   1:  PR[91,1] = PR[90,1] + 6.641;
   1:  PR[91,2] = PR[90,2] + -29.893;
   1:  PR[91,3] = PR[90,3] + 98.074;
   1:L PR[91] R[100]mm/sec CNT100;
   1:  PR[91,1] = PR[90,1] + 10.896;
   1:  PR[91,2] = PR[90,2] + -30.120;
   1:  PR[91,3] = PR[90,3] + 98.081;
   1:L PR[91] R[100]mm/sec CNT100;
   1:  PR[91,1] = PR[90,1] + 16.041;
   1:  PR[91,2] = PR[90,2] + -30.372;
   1:  PR[91,3] = PR[90,3] + 98.101;
   1:L PR[91] R[100]mm/sec CNT100;
   1:  PR[91,1] = PR[90,1] + 18.590;
   1:  PR[91,2] = PR[90,2] + -30.271;
   1:  PR[91,3] = PR[90,3] + 98.125;
   1:L PR[91] R[100]mm/sec CNT100;
   1:  PR[91,1] = PR[90,1] + 25.648;
   1:  PR[91,2] = PR[90,2] + -29.896;
   1:  PR[91,3] = PR[90,3] + 98.137;
   1:L PR[91] R[100]mm/sec CNT100;
   1:  PR[91,1] = PR[90,1] + 25.448;
   1:  PR[91,2] = PR[90,2] + -30.607;
   1:  PR[91,3] = PR[90,3] + 98.169;
   1:L PR[91] R[100]mm/sec CNT100;
   1:  PR[91,1] = PR[90,1] + 28.784;
   1:  PR[91,2] = PR[90,2] + -31.148;
   1:  PR[91,3] = PR[90,3] + 98.173;
   1:L PR[91] R[100]mm/sec CNT100;
   1:  PR[91,1] = PR[90,1] + 29.348;
   1:  PR[91,2] = PR[90,2] + -31.179;
   1:  PR[91,3] = PR[90,3] + 98.188;
   1:L PR[91] R[100]mm/sec CNT100;
   1:  PR[91,1] = PR[90,1] + 34.258;
   1:  PR[91,2] = PR[90,2] + -31.084;
   1:  PR[91,3] = PR[90,3] + 98.191;
   1:L PR[91] R[100]mm/sec CNT100;
   1:  PR[91,1] = PR[90,1] + 35.080;
   1:  PR[91,2] = PR[90,2] + -30.981;
   1:  PR[91,3] = PR[90,3] + 98.214;
   1:L PR[91] R[100]mm/sec CNT100;
   1:  PR[91,1] = PR[90,1] + 39.542;
   1:  PR[91,2] = PR[90,2] + -30.057;
   1:  PR[91,3] = PR[90,3] + 98.217;
   1:L PR[91] R[100]mm/sec CNT100;
   1:  PR[91,1] = PR[90,1] + 40.641;
   1:  PR[91,2] = PR[90,2] + -29.713;
   1:  PR[91,3] = PR[90,3] + 98.239;
   1:L PR[91] R[100]mm/sec CNT100;
   1:  PR[91,1] = PR[90,1] + 44.461;
   1:  PR[91,2] = PR[90,2] + -28.152;
   1:  PR[91,3] = PR[90,3] + 98.244;
   1:L PR[91] R[100]mm/sec CNT100;
   1:  PR[91,1] = PR[90,1] + 45.821;
   1:  PR[91,2] = PR[90,2] + -27.441;
   1:  PR[91,3] = PR[90,3] + 98.263;
   1:L PR[91] R[100]mm/sec CNT100;
   1:  PR[91,1] = PR[90,1] + 48.863;
   1:  PR[91,2] = PR[90,2] + -25.483;
   1:  PR[91,3] = PR[90,3] + 98.270;
   1:L PR[91] R[100]mm/sec CNT100;
   1:  PR[91,1] = PR[90,1] + 50.435;
   1:  PR[91,2] = PR[90,2] + -24.267;
   1:  PR[91,3] = PR[90,3] + 98.287;
   1:L PR[91] R[100]mm/sec CNT100;
   1:  PR[91,1] = PR[90,1] + 52.635;
   1:  PR[91,2] = PR[90,2] + -22.198;
   1:  PR[91,3] = PR[90,3] + 98.296;
   1:L PR[91] R[100]mm/sec CNT100;
   1:  PR[91,1] = PR[90,1] + 54.323;
   1:  PR[91,2] = PR[90,2] + -20.343;
   1:  PR[91,3] = PR[90,3] + 98.310;
   1:L PR[91] R[100]mm/sec CNT100;
   1:  PR[91,1] = PR[90,1] + 55.712;
   1:  PR[91,2] = PR[90,2] + -18.450;
   1:  PR[91,3] = PR[90,3] + 98.321;
   1:L PR[91] R[100]mm/sec CNT100;
   1:  PR[91,1] = PR[90,1] + 57.371;
   1:  PR[91,2] = PR[90,2] + -15.845;
   1:  PR[91,3] = PR[90,3] + 98.332;
   1:L PR[91] R[100]mm/sec CNT100;
   1:  PR[91,1] = PR[90,1] + 58.087;
   1:  PR[91,2] = PR[90,2] + -14.370;
   1:  PR[91,3] = PR[90,3] + 98.347;
   1:L PR[91] R[100]mm/sec CNT100;
   1:  PR[91,1] = PR[90,1] + 59.526;
   1:  PR[91,2] = PR[90,2] + -10.971;
   1:  PR[91,3] = PR[90,3] + 98.354;
   1:L PR[91] R[100]mm/sec CNT100;
   1:  PR[91,1] = PR[90,1] + 59.787;
   1:  PR[91,2] = PR[90,2] + -10.029;
   1:  PR[91,3] = PR[90,3] + 98.371;
   1:L PR[91] R[100]mm/sec CNT100;
   1:  PR[91,1] = PR[90,1] + 60.788;
   1:  PR[91,2] = PR[90,2] + -5.902;
   1:  PR[91,3] = PR[90,3] + 98.376;
   1:L PR[91] R[100]mm/sec CNT100;
   1:  PR[91,1] = PR[90,1] + 61.174;
   1:  PR[91,2] = PR[90,2] + -1.109;
   1:  PR[91,3] = PR[90,3] + 98.395;
   1:L PR[91] R[100]mm/sec CNT100;
   1:  PR[91,1] = PR[90,1] + 61.192;
   1:  PR[91,2] = PR[90,2] + -0.755;
   1:  PR[91,3] = PR[90,3] + 98.418;
   1:L PR[91] R[100]mm/sec CNT100;
   1:  PR[91,1] = PR[90,1] + 60.788;
   1:  PR[91,2] = PR[90,2] + 4.445;
   1:  PR[91,3] = PR[90,3] + 98.419;
   1:L PR[91] R[100]mm/sec CNT100;
   1:  PR[91,1] = PR[90,1] + 59.787;
   1:  PR[91,2] = PR[90,2] + 8.570;
   1:  PR[91,3] = PR[90,3] + 98.443;
   1:L PR[91] R[100]mm/sec CNT100;
   1:  PR[91,1] = PR[90,1] + 59.526;
   1:  PR[91,2] = PR[90,2] + 9.512;
   1:  PR[91,3] = PR[90,3] + 98.463;
   1:L PR[91] R[100]mm/sec CNT100;
   1:  PR[91,1] = PR[90,1] + 58.087;
   1:  PR[91,2] = PR[90,2] + 12.910;
   1:  PR[91,3] = PR[90,3] + 98.467;
   1:L PR[91] R[100]mm/sec CNT100;
   1:  PR[91,1] = PR[90,1] + 57.372;
   1:  PR[91,2] = PR[90,2] + 14.385;
   1:  PR[91,3] = PR[90,3] + 98.484;
   1:L PR[91] R[100]mm/sec CNT100;
   1:  PR[91,1] = PR[90,1] + 55.713;
   1:  PR[91,2] = PR[90,2] + 16.990;
   1:  PR[91,3] = PR[90,3] + 98.492;
   1:L PR[91] R[100]mm/sec CNT100;
   1:  PR[91,1] = PR[90,1] + 54.325;
   1:  PR[91,2] = PR[90,2] + 18.882;
   1:  PR[91,3] = PR[90,3] + 98.506;
   1:L PR[91] R[100]mm/sec CNT100;
   1:  PR[91,1] = PR[90,1] + 52.637;
   1:  PR[91,2] = PR[90,2] + 20.737;
   1:  PR[91,3] = PR[90,3] + 98.517;
   1:L PR[91] R[100]mm/sec CNT100;
   1:  PR[91,1] = PR[90,1] + 50.438;
   1:  PR[91,2] = PR[90,2] + 22.806;
   1:  PR[91,3] = PR[90,3] + 98.529;
   1:L PR[91] R[100]mm/sec CNT100;
   1:  PR[91,1] = PR[90,1] + 48.866;
   1:  PR[91,2] = PR[90,2] + 24.022;
   1:  PR[91,3] = PR[90,3] + 98.543;
   1:L PR[91] R[100]mm/sec CNT100;
   1:  PR[91,1] = PR[90,1] + 45.826;
   1:  PR[91,2] = PR[90,2] + 25.979;
   1:  PR[91,3] = PR[90,3] + 98.552;
   1:L PR[91] R[100]mm/sec CNT100;
   1:  PR[91,1] = PR[90,1] + 44.466;
   1:  PR[91,2] = PR[90,2] + 26.691;
   1:  PR[91,3] = PR[90,3] + 98.569;
   1:L PR[91] R[100]mm/sec CNT100;
   1:  PR[91,1] = PR[90,1] + 40.648;
   1:  PR[91,2] = PR[90,2] + 28.252;
   1:  PR[91,3] = PR[90,3] + 98.576;
   1:L PR[91] R[100]mm/sec CNT100;
   1:  PR[91,1] = PR[90,1] + 39.550;
   1:  PR[91,2] = PR[90,2] + 28.596;
   1:  PR[91,3] = PR[90,3] + 98.595;
   1:L PR[91] R[100]mm/sec CNT100;
   1:  PR[91,1] = PR[90,1] + 35.089;
   1:  PR[91,2] = PR[90,2] + 29.521;
   1:  PR[91,3] = PR[90,3] + 98.600;
   1:L PR[91] R[100]mm/sec CNT100;
   1:  PR[91,1] = PR[90,1] + 34.267;
   1:  PR[91,2] = PR[90,2] + 29.624;
   1:  PR[91,3] = PR[90,3] + 98.621;
   1:L PR[91] R[100]mm/sec CNT100;
   1:  PR[91,1] = PR[90,1] + 29.359;
   1:  PR[91,2] = PR[90,2] + 29.721;
   1:  PR[91,3] = PR[90,3] + 98.625;
   1:L PR[91] R[100]mm/sec CNT100;
   1:  PR[91,1] = PR[90,1] + 28.796;
   1:  PR[91,2] = PR[90,2] + 29.690;
   1:  PR[91,3] = PR[90,3] + 98.648;
   1:L PR[91] R[100]mm/sec CNT100;
   1:  PR[91,1] = PR[90,1] + 23.729;
   1:  PR[91,2] = PR[90,2] + 28.869;
   1:  PR[91,3] = PR[90,3] + 98.650;
   1:L PR[91] R[100]mm/sec CNT100;
   1:  PR[91,1] = PR[90,1] + 23.140;
   1:  PR[91,2] = PR[90,2] + 28.730;
   1:  PR[91,3] = PR[90,3] + 98.674;
   1:L PR[91] R[100]mm/sec CNT100;
   1:  PR[91,1] = PR[90,1] + 18.623;
   1:  PR[91,2] = PR[90,2] + 28.811;
   1:  PR[91,3] = PR[90,3] + 98.677;
   1:L PR[91] R[100]mm/sec CNT100;
   1:  PR[91,1] = PR[90,1] + 16.042;
   1:  PR[91,2] = PR[90,2] + 28.913;
   1:  PR[91,3] = PR[90,3] + 98.698;
   1:L PR[91] R[100]mm/sec CNT100;
   1:  PR[91,1] = PR[90,1] + 10.897;
   1:  PR[91,2] = PR[90,2] + 28.661;
   1:  PR[91,3] = PR[90,3] + 98.710;
   1:L PR[91] R[100]mm/sec CNT100;
   1:  PR[91,1] = PR[90,1] + 6.641;
   1:  PR[91,2] = PR[90,2] + 28.434;
   1:  PR[91,3] = PR[90,3] + 98.733;
   1:L PR[91] R[100]mm/sec CNT100;
   1:  PR[91,1] = PR[90,1] + 5.106;
   1:  PR[91,2] = PR[90,2] + 28.225;
   1:  PR[91,3] = PR[90,3] + 98.753;
   1:L PR[91] R[100]mm/sec CNT100;
   1:  PR[91,1] = PR[90,1] + -3.145;
   1:  PR[91,2] = PR[90,2] + 27.325;
   1:  PR[91,3] = PR[90,3] + 98.760;
   1:L PR[91] R[100]mm/sec CNT100;
   1:  PR[91,1] = PR[90,1] + -5.199;
   1:  PR[91,2] = PR[90,2] + 26.959;
   1:  PR[91,3] = PR[90,3] + 98.799;
   1:L PR[91] R[100]mm/sec CNT100;
   1:  PR[91,1] = PR[90,1] + -12.780;
   1:  PR[91,2] = PR[90,2] + 25.572;
   1:  PR[91,3] = PR[90,3] + 98.808;
   1:L PR[91] R[100]mm/sec CNT100;
   1:  PR[91,1] = PR[90,1] + -16.949;
   1:  PR[91,2] = PR[90,2] + 24.489;
   1:  PR[91,3] = PR[90,3] + 98.844;
   1:L PR[91] R[100]mm/sec CNT100;
   1:  PR[91,1] = PR[90,1] + -21.539;
   1:  PR[91,2] = PR[90,2] + 23.273;
   1:  PR[91,3] = PR[90,3] + 98.864;
   1:L PR[91] R[100]mm/sec CNT100;
   1:  PR[91,1] = PR[90,1] + -29.296;
   1:  PR[91,2] = PR[90,2] + 20.506;
   1:  PR[91,3] = PR[90,3] + 98.886;
   1:L PR[91] R[100]mm/sec CNT100;
   1:  PR[91,1] = PR[90,1] + -35.940;
   1:  PR[91,2] = PR[90,2] + 17.361;
   1:  PR[91,3] = PR[90,3] + 98.924;
   1:L PR[91] R[100]mm/sec CNT100;
   1:  PR[91,1] = PR[90,1] + -38.987;
   1:  PR[91,2] = PR[90,2] + 15.439;
   1:  PR[91,3] = PR[90,3] + 98.958;
   1:L PR[91] R[100]mm/sec CNT100;
   1:  PR[91,1] = PR[90,1] + -41.065;
   1:  PR[91,2] = PR[90,2] + 14.002;
   1:  PR[91,3] = PR[90,3] + 98.974;
   1:L PR[91] R[100]mm/sec CNT100;
   1:  PR[91,1] = PR[90,1] + -42.431;
   1:  PR[91,2] = PR[90,2] + 12.638;
   1:  PR[91,3] = PR[90,3] + 98.986;
   1:L PR[91] R[100]mm/sec CNT100;
   1:  PR[91] = PR[90];
   1:  PR[91,1] = PR[90,1] + -44.925;
   1:  PR[91,2] = PR[90,2] + 7.871;
   1:  PR[91,3] = PR[90,3] + 100.295;
   1:L PR[91] R[100]mm/sec CNT100;
   1:  PR[91,1] = PR[90,1] + -46.371;
   1:  PR[91,2] = PR[90,2] + 5.287;
   1:  PR[91,3] = PR[90,3] + 99.008;
   1:L PR[91] R[100]mm/sec CNT100;
   1:  PR[91,1] = PR[90,1] + -46.992;
   1:  PR[91,2] = PR[90,2] + 3.826;
   1:  PR[91,3] = PR[90,3] + 99.021;
   1:L PR[91] R[100]mm/sec CNT100;
   1:  PR[91,1] = PR[90,1] + -47.631;
   1:  PR[91,2] = PR[90,2] + 0.359;
   1:  PR[91,3] = PR[90,3] + 99.029;
   1:L PR[91] R[100]mm/sec CNT100;
   1:  PR[91,1] = PR[90,1] + -47.771;
   1:  PR[91,2] = PR[90,2] + -0.655;
   1:  PR[91,3] = PR[90,3] + 99.045;
   1:L PR[91] R[100]mm/sec CNT100;
   1:  PR[91,1] = PR[90,1] + -47.136;
   1:  PR[91,2] = PR[90,2] + -3.623;
   1:  PR[91,3] = PR[90,3] + 99.050;
   1:L PR[91] R[100]mm/sec CNT100;
   1:  PR[91,1] = PR[90,1] + -46.916;
   1:  PR[91,2] = PR[90,2] + -5.255;
   1:  PR[91,3] = PR[90,3] + 99.064;
   1:L PR[91] R[100]mm/sec CNT100;
   1:  PR[91,1] = PR[90,1] + -46.201;
   1:  PR[91,2] = PR[90,2] + -6.956;
   1:  PR[91,3] = PR[90,3] + 99.072;
   1:L PR[91] R[100]mm/sec CNT100;
   1:  PR[91,1] = PR[90,1] + -44.928;
   1:  PR[91,2] = PR[90,2] + -9.234;
   1:  PR[91,3] = PR[90,3] + 99.081;
   1:L PR[91] R[100]mm/sec CNT100;
   1:  PR[91,1] = PR[90,1] + -43.216;
   1:  PR[91,2] = PR[90,2] + -11.609;
   1:  PR[91,3] = PR[90,3] + 99.093;
   1:L PR[91] R[100]mm/sec CNT100;
   1:  PR[91,1] = PR[90,1] + -42.222;
   1:  PR[91,2] = PR[90,2] + -12.617;
   1:  PR[91,3] = PR[90,3] + 99.106;
   1:L PR[91] R[100]mm/sec CNT100;
   1:  PR[91,1] = PR[90,1] + -39.392;
   1:  PR[91,2] = PR[90,2] + -15.330;
   1:  PR[91,3] = PR[90,3] + 99.113;
   1:L PR[91] R[100]mm/sec CNT100;
   1:  PR[91,1] = PR[90,1] + -39.188;
   1:  PR[91,2] = PR[90,2] + -15.505;
   1:  PR[91,3] = PR[90,3] + 99.131;
   1:L PR[91] R[100]mm/sec CNT100;
   1:  PR[91,1] = PR[90,1] + -33.702;
   1:  PR[91,2] = PR[90,2] + -18.967;
   1:  PR[91,3] = PR[90,3] + 99.133;
   1:L PR[91] R[100]mm/sec CNT100;
   1:  PR[91,1] = PR[90,1] + -27.011;
   1:  PR[91,2] = PR[90,2] + -22.137;
   1:  PR[91,3] = PR[90,3] + 99.163;
   1:L PR[91] R[100]mm/sec CNT100;
   1:  PR[91,1] = PR[90,1] + -19.200;
   1:  PR[91,2] = PR[90,2] + -24.928;
   1:  PR[91,3] = PR[90,3] + 99.197;
   1:L PR[91] R[100]mm/sec CNT100;
   1:  PR[91,1] = PR[90,1] + -13.832;
   1:  PR[91,2] = PR[90,2] + -26.349;
   1:  PR[91,3] = PR[90,3] + 99.236;
   1:L PR[91] R[100]mm/sec CNT100;
   1:  PR[91,1] = PR[90,1] + -10.380;
   1:  PR[91,2] = PR[90,2] + -27.246;
   1:  PR[91,3] = PR[90,3] + 99.262;
   1:L PR[91] R[100]mm/sec CNT100;
   1:  PR[91,1] = PR[90,1] + -0.670;
   1:  PR[91,2] = PR[90,2] + -29.016;
   1:  PR[91,3] = PR[90,3] + 99.279;
   1:L PR[91] R[100]mm/sec CNT100;
   1:  PR[91,1] = PR[90,1] + 4.458;
   1:  PR[91,2] = PR[90,2] + -29.576;
   1:  PR[91,3] = PR[90,3] + 99.325;
   1:L PR[91] R[100]mm/sec CNT100;
   1:  PR[91,1] = PR[90,1] + 8.317;
   1:  PR[91,2] = PR[90,2] + -30.101;
   1:  PR[91,3] = PR[90,3] + 99.349;
   1:L PR[91] R[100]mm/sec CNT100;
   1:  PR[91,1] = PR[90,1] + 18.123;
   1:  PR[91,2] = PR[90,2] + -30.626;
   1:  PR[91,3] = PR[90,3] + 99.367;
   1:L PR[91] R[100]mm/sec CNT100;
   1:  PR[91,1] = PR[90,1] + 26.250;
   1:  PR[91,2] = PR[90,2] + -30.195;
   1:  PR[91,3] = PR[90,3] + 99.413;
   1:L PR[91] R[100]mm/sec CNT100;
   1:  PR[91,1] = PR[90,1] + 26.060;
   1:  PR[91,2] = PR[90,2] + -30.872;
   1:  PR[91,3] = PR[90,3] + 99.451;
   1:L PR[91] R[100]mm/sec CNT100;
   1:  PR[91,1] = PR[90,1] + 28.993;
   1:  PR[91,2] = PR[90,2] + -31.346;
   1:  PR[91,3] = PR[90,3] + 99.454;
   1:L PR[91] R[100]mm/sec CNT100;
   1:  PR[91,1] = PR[90,1] + 34.620;
   1:  PR[91,2] = PR[90,2] + -31.231;
   1:  PR[91,3] = PR[90,3] + 99.468;
   1:L PR[91] R[100]mm/sec CNT100;
   1:  PR[91,1] = PR[90,1] + 40.124;
   1:  PR[91,2] = PR[90,2] + -30.092;
   1:  PR[91,3] = PR[90,3] + 99.494;
   1:L PR[91] R[100]mm/sec CNT100;
   1:  PR[91,1] = PR[90,1] + 40.146;
   1:  PR[91,2] = PR[90,2] + -30.085;
   1:  PR[91,3] = PR[90,3] + 99.521;
   1:L PR[91] R[100]mm/sec CNT100;
   1:  PR[91,1] = PR[90,1] + 45.193;
   1:  PR[91,2] = PR[90,2] + -28.023;
   1:L PR[91] R[100]mm/sec CNT100;
   1:  PR[91,1] = PR[90,1] + 45.424;
   1:  PR[91,2] = PR[90,2] + -27.902;
   1:  PR[91,3] = PR[90,3] + 99.546;
   1:L PR[91] R[100]mm/sec CNT100;
   1:  PR[91,1] = PR[90,1] + 49.743;
   1:  PR[91,2] = PR[90,2] + -25.122;
   1:  PR[91,3] = PR[90,3] + 99.547;
   1:L PR[91] R[100]mm/sec CNT100;
   1:  PR[91,1] = PR[90,1] + 50.169;
   1:  PR[91,2] = PR[90,2] + -24.793;
   1:  PR[91,3] = PR[90,3] + 99.571;
   1:L PR[91] R[100]mm/sec CNT100;
   1:  PR[91,1] = PR[90,1] + 53.644;
   1:  PR[91,2] = PR[90,2] + -21.525;
   1:  PR[91,3] = PR[90,3] + 99.574;
   1:L PR[91] R[100]mm/sec CNT100;
   1:  PR[91,1] = PR[90,1] + 54.218;
   1:  PR[91,2] = PR[90,2] + -20.895;
   1:  PR[91,3] = PR[90,3] + 99.596;
   1:L PR[91] R[100]mm/sec CNT100;
   1:  PR[91,1] = PR[90,1] + 56.802;
   1:  PR[91,2] = PR[90,2] + -17.374;
   1:  PR[91,3] = PR[90,3] + 99.600;
   1:L PR[91] R[100]mm/sec CNT100;
   1:  PR[91,1] = PR[90,1] + 57.445;
   1:  PR[91,2] = PR[90,2] + -16.364;
   1:  PR[91,3] = PR[90,3] + 99.620;
   1:L PR[91] R[100]mm/sec CNT100;
   1:  PR[91,1] = PR[90,1] + 59.170;
   1:  PR[91,2] = PR[90,2] + -12.806;
   1:  PR[91,3] = PR[90,3] + 99.626;
   1:L PR[91] R[100]mm/sec CNT100;
   1:  PR[91,1] = PR[90,1] + 59.773;
   1:  PR[91,2] = PR[90,2] + -11.383;
   1:  PR[91,3] = PR[90,3] + 99.645;
   1:L PR[91] R[100]mm/sec CNT100;
   1:  PR[91,1] = PR[90,1] + 60.727;
   1:  PR[91,2] = PR[90,2] + -7.931;
   1:  PR[91,3] = PR[90,3] + 99.652;
   1:L PR[91] R[100]mm/sec CNT100;
   1:  PR[91,1] = PR[90,1] + 61.163;
   1:  PR[91,2] = PR[90,2] + -6.135;
   1:  PR[91,3] = PR[90,3] + 99.668;
   1:L PR[91] R[100]mm/sec CNT100;
   1:  PR[91,1] = PR[90,1] + 61.350;
   1:  PR[91,2] = PR[90,2] + -3.722;
   1:  PR[91,3] = PR[90,3] + 99.677;
   1:L PR[91] R[100]mm/sec CNT100;
   1:  PR[91,1] = PR[90,1] + 61.612;
   1:  PR[91,2] = PR[90,2] + -0.718;
   1:  PR[91,3] = PR[90,3] + 99.688;
   1:L PR[91] R[100]mm/sec CNT100;
   1:  PR[91,1] = PR[90,1] + 61.475;
   1:  PR[91,2] = PR[90,2] + 1.093;
   1:  PR[91,3] = PR[90,3] + 99.702;
   1:L PR[91] R[100]mm/sec CNT100;
   1:  PR[91,1] = PR[90,1] + 61.166;
   1:  PR[91,2] = PR[90,2] + 4.666;
   1:  PR[91,3] = PR[90,3] + 99.711;
   1:L PR[91] R[100]mm/sec CNT100;
   1:  PR[91,1] = PR[90,1] + 60.727;
   1:  PR[91,2] = PR[90,2] + 6.472;
   1:  PR[91,3] = PR[90,3] + 99.728;
   1:L PR[91] R[100]mm/sec CNT100;
   1:  PR[91,1] = PR[90,1] + 59.774;
   1:  PR[91,2] = PR[90,2] + 9.922;
   1:  PR[91,3] = PR[90,3] + 99.736;
   1:L PR[91] R[100]mm/sec CNT100;
   1:  PR[91,1] = PR[90,1] + 59.171;
   1:  PR[91,2] = PR[90,2] + 11.346;
   1:  PR[91,3] = PR[90,3] + 99.753;
   1:L PR[91] R[100]mm/sec CNT100;
   1:  PR[91,1] = PR[90,1] + 57.446;
   1:  PR[91,2] = PR[90,2] + 14.902;
   1:  PR[91,3] = PR[90,3] + 99.760;
   1:L PR[91] R[100]mm/sec CNT100;
   1:  PR[91,1] = PR[90,1] + 56.803;
   1:  PR[91,2] = PR[90,2] + 15.912;
   1:  PR[91,3] = PR[90,3] + 99.779;
   1:L PR[91] R[100]mm/sec CNT100;
   1:  PR[91,1] = PR[90,1] + 54.221;
   1:  PR[91,2] = PR[90,2] + 19.433;
   1:  PR[91,3] = PR[90,3] + 99.784;
   1:L PR[91] R[100]mm/sec CNT100;
   1:  PR[91,1] = PR[90,1] + 53.647;
   1:  PR[91,2] = PR[90,2] + 20.063;
   1:  PR[91,3] = PR[90,3] + 99.805;
   1:L PR[91] R[100]mm/sec CNT100;
   1:  PR[91,1] = PR[90,1] + 50.174;
   1:  PR[91,2] = PR[90,2] + 23.330;
   1:  PR[91,3] = PR[90,3] + 99.809;
   1:L PR[91] R[100]mm/sec CNT100;
   1:  PR[91,1] = PR[90,1] + 49.748;
   1:  PR[91,2] = PR[90,2] + 23.660;
   1:  PR[91,3] = PR[90,3] + 99.831;
   1:L PR[91] R[100]mm/sec CNT100;
   1:  PR[91,1] = PR[90,1] + 45.431;
   1:  PR[91,2] = PR[90,2] + 26.439;
   1:  PR[91,3] = PR[90,3] + 99.833;
   1:L PR[91] R[100]mm/sec CNT100;
   1:  PR[91,1] = PR[90,1] + 45.200;
   1:  PR[91,2] = PR[90,2] + 26.560;
   1:  PR[91,3] = PR[90,3] + 99.857;
   1:L PR[91] R[100]mm/sec CNT100;
   1:  PR[91,1] = PR[90,1] + 40.155;
   1:  PR[91,2] = PR[90,2] + 28.623;
   1:  PR[91,3] = PR[90,3] + 99.859;
   1:L PR[91] R[100]mm/sec CNT100;
   1:  PR[91,1] = PR[90,1] + 40.133;
   1:  PR[91,2] = PR[90,2] + 28.630;
   1:  PR[91,3] = PR[90,3] + 99.884;
   1:L PR[91] R[100]mm/sec CNT100;
   1:  PR[91,1] = PR[90,1] + 34.626;
   1:  PR[91,2] = PR[90,2] + 29.771;
   1:L PR[91] R[100]mm/sec CNT100;
   1:  PR[91,1] = PR[90,1] + 29.012;
   1:  PR[91,2] = PR[90,2] + 29.888;
   1:  PR[91,3] = PR[90,3] + 99.910;
   1:L PR[91] R[100]mm/sec CNT100;
   1:  PR[91,1] = PR[90,1] + 28.964;
   1:  PR[91,2] = PR[90,2] + 29.884;
   1:  PR[91,3] = PR[90,3] + 99.937;
   1:L PR[91] R[100]mm/sec CNT100;
   1:  PR[91,1] = PR[90,1] + 23.663;
   1:  PR[91,2] = PR[90,2] + 29.025;
   1:L PR[91] R[100]mm/sec CNT100;
   1:  PR[91,1] = PR[90,1] + 18.121;
   1:  PR[91,2] = PR[90,2] + 29.168;
   1:  PR[91,3] = PR[90,3] + 99.962;
   1:L PR[91] R[100]mm/sec CNT100;
   1:  PR[91,1] = PR[90,1] + 8.318;
   1:  PR[91,2] = PR[90,2] + 28.642;
   1:  PR[91,3] = PR[90,3] + 99.988;
   1:L PR[91] R[100]mm/sec CNT100;
   1:  PR[91,1] = PR[90,1] + 4.458;
   1:  PR[91,2] = PR[90,2] + 28.117;
   1:  PR[91,3] = PR[90,3] + 100.034;
   1:L PR[91] R[100]mm/sec CNT100;
   1:  PR[91,1] = PR[90,1] + -0.670;
   1:  PR[91,2] = PR[90,2] + 27.557;
   1:  PR[91,3] = PR[90,3] + 100.052;
   1:L PR[91] R[100]mm/sec CNT100;
   1:  PR[91,1] = PR[90,1] + -10.380;
   1:  PR[91,2] = PR[90,2] + 25.788;
   1:  PR[91,3] = PR[90,3] + 100.076;
   1:L PR[91] R[100]mm/sec CNT100;
   1:  PR[91,1] = PR[90,1] + -13.831;
   1:  PR[91,2] = PR[90,2] + 24.891;
   1:  PR[91,3] = PR[90,3] + 100.122;
   1:L PR[91] R[100]mm/sec CNT100;
   1:  PR[91,1] = PR[90,1] + -19.200;
   1:  PR[91,2] = PR[90,2] + 23.469;
   1:  PR[91,3] = PR[90,3] + 100.139;
   1:L PR[91] R[100]mm/sec CNT100;
   1:  PR[91,1] = PR[90,1] + -27.011;
   1:  PR[91,2] = PR[90,2] + 20.679;
   1:  PR[91,3] = PR[90,3] + 100.165;
   1:L PR[91] R[100]mm/sec CNT100;
   1:  PR[91,1] = PR[90,1] + -33.702;
   1:  PR[91,2] = PR[90,2] + 17.508;
   1:  PR[91,3] = PR[90,3] + 100.203;
   1:L PR[91] R[100]mm/sec CNT100;
   1:  PR[91,1] = PR[90,1] + -39.188;
   1:  PR[91,2] = PR[90,2] + 14.047;
   1:  PR[91,3] = PR[90,3] + 100.238;
   1:L PR[91] R[100]mm/sec CNT100;
   1:  PR[91,1] = PR[90,1] + -39.388;
   1:  PR[91,2] = PR[90,2] + 13.874;
   1:  PR[91,3] = PR[90,3] + 100.268;
   1:L PR[91] R[100]mm/sec CNT100;
   1:  PR[91,1] = PR[90,1] + -43.328;
   1:  PR[91,2] = PR[90,2] + 10.061;
   1:  PR[91,3] = PR[90,3] + 100.269;
   1:L PR[91] R[100]mm/sec CNT100;
   1:  PR[91] = PR[90];
   1:  PR[91,1] = PR[90,1] + -43.344;
   1:  PR[91,2] = PR[90,2] + 7.465;
   1:  PR[91,3] = PR[90,3] + 101.595;
   1:L PR[91] R[100]mm/sec CNT100;
   1:  PR[91,1] = PR[90,1] + -44.199;
   1:  PR[91,2] = PR[90,2] + 5.937;
   1:  PR[91,3] = PR[90,3] + 100.312;
   1:L PR[91] R[100]mm/sec CNT100;
   1:  PR[91,1] = PR[90,1] + -45.194;
   1:  PR[91,2] = PR[90,2] + 3.593;
   1:  PR[91,3] = PR[90,3] + 100.321;
   1:L PR[91] R[100]mm/sec CNT100;
   1:  PR[91,1] = PR[90,1] + -45.628;
   1:  PR[91,2] = PR[90,2] + 1.240;
   1:  PR[91,3] = PR[90,3] + 100.333;
   1:L PR[91] R[100]mm/sec CNT100;
   1:  PR[91,1] = PR[90,1] + -45.891;
   1:  PR[91,2] = PR[90,2] + -0.655;
   1:  PR[91,3] = PR[90,3] + 100.344;
   1:L PR[91] R[100]mm/sec CNT100;
   1:  PR[91,1] = PR[90,1] + -45.449;
   1:  PR[91,2] = PR[90,2] + -2.720;
   1:  PR[91,3] = PR[90,3] + 100.353;
   1:L PR[91] R[100]mm/sec CNT100;
   1:  PR[91,1] = PR[90,1] + -45.135;
   1:  PR[91,2] = PR[90,2] + -5.045;
   1:  PR[91,3] = PR[90,3] + 100.363;
   1:L PR[91] R[100]mm/sec CNT100;
   1:  PR[91,1] = PR[90,1] + -44.092;
   1:  PR[91,2] = PR[90,2] + -7.528;
   1:  PR[91,3] = PR[90,3] + 100.374;
   1:L PR[91] R[100]mm/sec CNT100;
   1:  PR[91,1] = PR[90,1] + -43.344;
   1:  PR[91,2] = PR[90,2] + -8.866;
   1:  PR[91,3] = PR[90,3] + 100.387;
   1:L PR[91] R[100]mm/sec CNT100;
   1:  PR[91,1] = PR[90,1] + -41.134;
   1:  PR[91,2] = PR[90,2] + -11.932;
   1:  PR[91,3] = PR[90,3] + 100.394;
   1:L PR[91] R[100]mm/sec CNT100;
   1:  PR[91,1] = PR[90,1] + -40.904;
   1:  PR[91,2] = PR[90,2] + -12.166;
   1:  PR[91,3] = PR[90,3] + 100.412;
   1:L PR[91] R[100]mm/sec CNT100;
   1:  PR[91,1] = PR[90,1] + -40.040;
   1:  PR[91,2] = PR[90,2] + -12.993;
   1:  PR[91,3] = PR[90,3] + 100.413;
   1:L PR[91] R[100]mm/sec CNT100;
   1:  PR[91,1] = PR[90,1] + -36.989;
   1:  PR[91,2] = PR[90,2] + -15.626;
   1:  PR[91,3] = PR[90,3] + 100.419;
   1:L PR[91] R[100]mm/sec CNT100;
   1:  PR[91,1] = PR[90,1] + -31.464;
   1:  PR[91,2] = PR[90,2] + -19.115;
   1:  PR[91,3] = PR[90,3] + 100.438;
   1:L PR[91] R[100]mm/sec CNT100;
   1:  PR[91,1] = PR[90,1] + -24.726;
   1:  PR[91,2] = PR[90,2] + -22.310;
   1:  PR[91,3] = PR[90,3] + 100.469;
   1:L PR[91] R[100]mm/sec CNT100;
   1:  PR[91,1] = PR[90,1] + -16.862;
   1:  PR[91,2] = PR[90,2] + -25.123;
   1:  PR[91,3] = PR[90,3] + 100.504;
   1:L PR[91] R[100]mm/sec CNT100;
   1:  PR[91,1] = PR[90,1] + -7.975;
   1:  PR[91,2] = PR[90,2] + -27.463;
   1:  PR[91,3] = PR[90,3] + 100.543;
   1:L PR[91] R[100]mm/sec CNT100;
   1:  PR[91,1] = PR[90,1] + 1.801;
   1:  PR[91,2] = PR[90,2] + -29.248;
   1:  PR[91,3] = PR[90,3] + 100.586;
   1:L PR[91] R[100]mm/sec CNT100;
   1:  PR[91,1] = PR[90,1] + 3.810;
   1:  PR[91,2] = PR[90,2] + -29.467;
   1:  PR[91,3] = PR[90,3] + 100.633;
   1:L PR[91] R[100]mm/sec CNT100;
   1:  PR[91,1] = PR[90,1] + 9.993;
   1:  PR[91,2] = PR[90,2] + -30.309;
   1:  PR[91,3] = PR[90,3] + 100.643;
   1:L PR[91] R[100]mm/sec CNT100;
   1:  PR[91,1] = PR[90,1] + 17.071;
   1:  PR[91,2] = PR[90,2] + -30.686;
   1:  PR[91,3] = PR[90,3] + 100.672;
   1:L PR[91] R[100]mm/sec CNT100;
   1:  PR[91,1] = PR[90,1] + 19.711;
   1:  PR[91,2] = PR[90,2] + -30.859;
   1:  PR[91,3] = PR[90,3] + 100.706;
   1:L PR[91] R[100]mm/sec CNT100;
   1:  PR[91,1] = PR[90,1] + 19.899;
   1:  PR[91,2] = PR[90,2] + -30.862;
   1:  PR[91,3] = PR[90,3] + 100.718;
   1:L PR[91] R[100]mm/sec CNT100;
   1:  PR[91,1] = PR[90,1] + 26.852;
   1:  PR[91,2] = PR[90,2] + -30.493;
   1:  PR[91,3] = PR[90,3] + 100.719;
   1:L PR[91] R[100]mm/sec CNT100;
   1:  PR[91,1] = PR[90,1] + 26.671;
   1:  PR[91,2] = PR[90,2] + -31.138;
   1:  PR[91,3] = PR[90,3] + 100.752;
   1:L PR[91] R[100]mm/sec CNT100;
   1:  PR[91,1] = PR[90,1] + 28.452;
   1:  PR[91,2] = PR[90,2] + -31.427;
   1:  PR[91,3] = PR[90,3] + 100.755;
   1:L PR[91] R[100]mm/sec CNT100;
   1:  PR[91,1] = PR[90,1] + 28.695;
   1:  PR[91,2] = PR[90,2] + -31.455;
   1:  PR[91,3] = PR[90,3] + 100.764;
   1:L PR[91] R[100]mm/sec CNT100;
   1:  PR[91,1] = PR[90,1] + 29.671;
   1:  PR[91,2] = PR[90,2] + -31.519;
   1:  PR[91,3] = PR[90,3] + 100.765;
   1:L PR[91] R[100]mm/sec CNT100;
   1:  PR[91,1] = PR[90,1] + 34.356;
   1:  PR[91,2] = PR[90,2] + -31.423;
   1:  PR[91,3] = PR[90,3] + 100.769;
   1:L PR[91] R[100]mm/sec CNT100;
   1:  PR[91,1] = PR[90,1] + 35.246;
   1:  PR[91,2] = PR[90,2] + -31.332;
   1:  PR[91,3] = PR[90,3] + 100.791;
   1:L PR[91] R[100]mm/sec CNT100;
   1:  PR[91,1] = PR[90,1] + 39.887;
   1:  PR[91,2] = PR[90,2] + -30.361;
   1:  PR[91,3] = PR[90,3] + 100.796;
   1:L PR[91] R[100]mm/sec CNT100;
   1:  PR[91,1] = PR[90,1] + 40.682;
   1:  PR[91,2] = PR[90,2] + -30.139;
   1:  PR[91,3] = PR[90,3] + 100.818;
   1:L PR[91] R[100]mm/sec CNT100;
   1:  PR[91,1] = PR[90,1] + 45.128;
   1:  PR[91,2] = PR[90,2] + -28.305;
   1:  PR[91,3] = PR[90,3] + 100.822;
   1:L PR[91] R[100]mm/sec CNT100;
   1:  PR[91,1] = PR[90,1] + 45.801;
   1:  PR[91,2] = PR[90,2] + -27.987;
   1:  PR[91,3] = PR[90,3] + 100.845;
   1:L PR[91] R[100]mm/sec CNT100;
   1:  PR[91,1] = PR[90,1] + 49.908;
   1:  PR[91,2] = PR[90,2] + -25.320;
   1:  PR[91,3] = PR[90,3] + 100.848;
   1:L PR[91] R[100]mm/sec CNT100;
   1:  PR[91,1] = PR[90,1] + 50.441;
   1:  PR[91,2] = PR[90,2] + -24.946;
   1:  PR[91,3] = PR[90,3] + 100.871;
   1:L PR[91] R[100]mm/sec CNT100;
   1:  PR[91,1] = PR[90,1] + 54.067;
   1:  PR[91,2] = PR[90,2] + -21.507;
   1:  PR[91,3] = PR[90,3] + 100.874;
   1:L PR[91] R[100]mm/sec CNT100;
   1:  PR[91,1] = PR[90,1] + 54.453;
   1:  PR[91,2] = PR[90,2] + -21.125;
   1:  PR[91,3] = PR[90,3] + 100.898;
   1:L PR[91] R[100]mm/sec CNT100;
   1:  PR[91,1] = PR[90,1] + 57.716;
   1:  PR[91,2] = PR[90,2] + -16.629;
   1:  PR[91,3] = PR[90,3] + 100.900;
   1:L PR[91] R[100]mm/sec CNT100;
   1:  PR[91,1] = PR[90,1] + 60.117;
   1:  PR[91,2] = PR[90,2] + -11.632;
   1:  PR[91,3] = PR[90,3] + 100.927;
   1:L PR[91] R[100]mm/sec CNT100;
   1:  PR[91,1] = PR[90,1] + 61.589;
   1:  PR[91,2] = PR[90,2] + -6.270;
   1:  PR[91,3] = PR[90,3] + 100.953;
   1:L PR[91] R[100]mm/sec CNT100;
   1:  PR[91,1] = PR[90,1] + 62.101;
   1:  PR[91,2] = PR[90,2] + -0.729;
   1:  PR[91,3] = PR[90,3] + 100.979;
   1:L PR[91] R[100]mm/sec CNT100;
   1:  PR[91,1] = PR[90,1] + 61.589;
   1:  PR[91,2] = PR[90,2] + 4.810;
   1:  PR[91,3] = PR[90,3] + 101.005;
   1:L PR[91] R[100]mm/sec CNT100;
   1:  PR[91,1] = PR[90,1] + 60.117;
   1:  PR[91,2] = PR[90,2] + 10.174;
   1:  PR[91,3] = PR[90,3] + 101.031;
   1:L PR[91] R[100]mm/sec CNT100;
   1:  PR[91,1] = PR[90,1] + 59.976;
   1:  PR[91,2] = PR[90,2] + 10.471;
   1:  PR[91,3] = PR[90,3] + 101.058;
   1:L PR[91] R[100]mm/sec CNT100;
   1:  PR[91,1] = PR[90,1] + 57.718;
   1:  PR[91,2] = PR[90,2] + 15.167;
   1:  PR[91,3] = PR[90,3] + 101.059;
   1:L PR[91] R[100]mm/sec CNT100;
   1:  PR[91,1] = PR[90,1] + 54.455;
   1:  PR[91,2] = PR[90,2] + 19.663;
   1:  PR[91,3] = PR[90,3] + 101.084;
   1:L PR[91] R[100]mm/sec CNT100;
   1:  PR[91,1] = PR[90,1] + 54.070;
   1:  PR[91,2] = PR[90,2] + 20.045;
   1:  PR[91,3] = PR[90,3] + 101.110;
   1:L PR[91] R[100]mm/sec CNT100;
   1:  PR[91,1] = PR[90,1] + 50.445;
   1:  PR[91,2] = PR[90,2] + 23.485;
   1:  PR[91,3] = PR[90,3] + 101.112;
   1:L PR[91] R[100]mm/sec CNT100;
   1:  PR[91,1] = PR[90,1] + 49.912;
   1:  PR[91,2] = PR[90,2] + 23.858;
   1:  PR[91,3] = PR[90,3] + 101.136;
   1:L PR[91] R[100]mm/sec CNT100;
   1:  PR[91,1] = PR[90,1] + 45.805;
   1:  PR[91,2] = PR[90,2] + 26.526;
   1:  PR[91,3] = PR[90,3] + 101.139;
   1:L PR[91] R[100]mm/sec CNT100;
   1:  PR[91,1] = PR[90,1] + 45.133;
   1:  PR[91,2] = PR[90,2] + 26.844;
   1:  PR[91,3] = PR[90,3] + 101.162;
   1:L PR[91] R[100]mm/sec CNT100;
   1:  PR[91,1] = PR[90,1] + 40.687;
   1:  PR[91,2] = PR[90,2] + 28.679;
   1:  PR[91,3] = PR[90,3] + 101.166;
   1:L PR[91] R[100]mm/sec CNT100;
   1:  PR[91,1] = PR[90,1] + 39.892;
   1:  PR[91,2] = PR[90,2] + 28.900;
   1:  PR[91,3] = PR[90,3] + 101.188;
   1:L PR[91] R[100]mm/sec CNT100;
   1:  PR[91,1] = PR[90,1] + 35.251;
   1:  PR[91,2] = PR[90,2] + 29.873;
   1:  PR[91,3] = PR[90,3] + 101.192;
   1:L PR[91] R[100]mm/sec CNT100;
   1:  PR[91,1] = PR[90,1] + 34.362;
   1:  PR[91,2] = PR[90,2] + 29.964;
   1:  PR[91,3] = PR[90,3] + 101.215;
   1:L PR[91] R[100]mm/sec CNT100;
   1:  PR[91,1] = PR[90,1] + 29.677;
   1:  PR[91,2] = PR[90,2] + 30.061;
   1:  PR[91,3] = PR[90,3] + 101.219;
   1:L PR[91] R[100]mm/sec CNT100;
   1:  PR[91,1] = PR[90,1] + 28.703;
   1:  PR[91,2] = PR[90,2] + 29.996;
   1:  PR[91,3] = PR[90,3] + 101.241;
   1:L PR[91] R[100]mm/sec CNT100;
   1:  PR[91,1] = PR[90,1] + 28.411;
   1:  PR[91,2] = PR[90,2] + 29.962;
   1:  PR[91,3] = PR[90,3] + 101.245;
   1:L PR[91] R[100]mm/sec CNT100;
   1:  PR[91,1] = PR[90,1] + 24.273;
   1:  PR[91,2] = PR[90,2] + 29.292;
   1:  PR[91,3] = PR[90,3] + 101.247;
   1:L PR[91] R[100]mm/sec CNT100;
   1:  PR[91,1] = PR[90,1] + 19.975;
   1:  PR[91,2] = PR[90,2] + 29.404;
   1:  PR[91,3] = PR[90,3] + 101.267;
   1:L PR[91] R[100]mm/sec CNT100;
   1:  PR[91,1] = PR[90,1] + 19.713;
   1:  PR[91,2] = PR[90,2] + 29.400;
   1:  PR[91,3] = PR[90,3] + 101.287;
   1:L PR[91] R[100]mm/sec CNT100;
   1:  PR[91,1] = PR[90,1] + 17.071;
   1:  PR[91,2] = PR[90,2] + 29.227;
   1:  PR[91,3] = PR[90,3] + 101.288;
   1:L PR[91] R[100]mm/sec CNT100;
   1:  PR[91,1] = PR[90,1] + 9.994;
   1:  PR[91,2] = PR[90,2] + 28.850;
   1:  PR[91,3] = PR[90,3] + 101.301;
   1:L PR[91] R[100]mm/sec CNT100;
   1:  PR[91,1] = PR[90,1] + 3.810;
   1:  PR[91,2] = PR[90,2] + 28.009;
   1:  PR[91,3] = PR[90,3] + 101.334;
   1:L PR[91] R[100]mm/sec CNT100;
   1:  PR[91,1] = PR[90,1] + 1.801;
   1:  PR[91,2] = PR[90,2] + 27.789;
   1:  PR[91,3] = PR[90,3] + 101.363;
   1:L PR[91] R[100]mm/sec CNT100;
   1:  PR[91,1] = PR[90,1] + -7.978;
   1:  PR[91,2] = PR[90,2] + 26.003;
   1:  PR[91,3] = PR[90,3] + 101.373;
   1:L PR[91] R[100]mm/sec CNT100;
   1:  PR[91,1] = PR[90,1] + -10.714;
   1:  PR[91,2] = PR[90,2] + 25.292;
   1:  PR[91,3] = PR[90,3] + 101.420;
   1:L PR[91] R[100]mm/sec CNT100;
   1:  PR[91,1] = PR[90,1] + -16.860;
   1:  PR[91,2] = PR[90,2] + 23.665;
   1:  PR[91,3] = PR[90,3] + 101.433;
   1:L PR[91] R[100]mm/sec CNT100;
   1:  PR[91,1] = PR[90,1] + -24.726;
   1:  PR[91,2] = PR[90,2] + 20.852;
   1:  PR[91,3] = PR[90,3] + 101.463;
   1:L PR[91] R[100]mm/sec CNT100;
   1:  PR[91,1] = PR[90,1] + -31.465;
   1:  PR[91,2] = PR[90,2] + 17.656;
   1:  PR[91,3] = PR[90,3] + 101.503;
   1:L PR[91] R[100]mm/sec CNT100;
   1:  PR[91,1] = PR[90,1] + -36.596;
   1:  PR[91,2] = PR[90,2] + 14.418;
   1:  PR[91,3] = PR[90,3] + 101.538;
   1:L PR[91] R[100]mm/sec CNT100;
   1:  PR[91,1] = PR[90,1] + -36.985;
   1:  PR[91,2] = PR[90,2] + 14.170;
   1:  PR[91,3] = PR[90,3] + 101.566;
   1:L PR[91] R[100]mm/sec CNT100;
   1:  PR[91,1] = PR[90,1] + -40.036;
   1:  PR[91,2] = PR[90,2] + 11.538;
   1:  PR[91,3] = PR[90,3] + 101.568;
   1:L PR[91] R[100]mm/sec CNT100;
   1:  PR[91,1] = PR[90,1] + -41.182;
   1:  PR[91,2] = PR[90,2] + 10.429;
   1:  PR[91,3] = PR[90,3] + 101.587;
   1:L PR[91] R[100]mm/sec CNT100;
   1:  PR[91] = PR[90];
   1:  PR[91,1] = PR[90,1] + -41.762;
   1:  PR[91,2] = PR[90,2] + 7.058;
   1:  PR[91,3] = PR[90,3] + 102.895;
   1:L PR[91] R[100]mm/sec CNT100;
   1:  PR[91,1] = PR[90,1] + -42.026;
   1:  PR[91,2] = PR[90,2] + 6.587;
   1:  PR[91,3] = PR[90,3] + 101.606;
   1:L PR[91] R[100]mm/sec CNT100;
   1:  PR[91,1] = PR[90,1] + -43.397;
   1:  PR[91,2] = PR[90,2] + 3.360;
   1:  PR[91,3] = PR[90,3] + 101.608;
   1:L PR[91] R[100]mm/sec CNT100;
   1:  PR[91,1] = PR[90,1] + -43.625;
   1:  PR[91,2] = PR[90,2] + 2.121;
   1:  PR[91,3] = PR[90,3] + 101.625;
   1:L PR[91] R[100]mm/sec CNT100;
   1:  PR[91,1] = PR[90,1] + -44.011;
   1:  PR[91,2] = PR[90,2] + -0.655;
   1:  PR[91,3] = PR[90,3] + 101.631;
   1:L PR[91] R[100]mm/sec CNT100;
   1:  PR[91,1] = PR[90,1] + -43.762;
   1:  PR[91,2] = PR[90,2] + -1.816;
   1:  PR[91,3] = PR[90,3] + 101.644;
   1:L PR[91] R[100]mm/sec CNT100;
   1:  PR[91,1] = PR[90,1] + -43.354;
   1:  PR[91,2] = PR[90,2] + -4.835;
   1:  PR[91,3] = PR[90,3] + 101.650;
   1:L PR[91] R[100]mm/sec CNT100;
   1:  PR[91,1] = PR[90,1] + -41.983;
   1:  PR[91,2] = PR[90,2] + -8.100;
   1:  PR[91,3] = PR[90,3] + 101.664;
   1:L PR[91] R[100]mm/sec CNT100;
   1:  PR[91,1] = PR[90,1] + -41.761;
   1:  PR[91,2] = PR[90,2] + -8.498;
   1:  PR[91,3] = PR[90,3] + 101.681;
   1:L PR[91] R[100]mm/sec CNT100;
   1:  PR[91,1] = PR[90,1] + -40.439;
   1:  PR[91,2] = PR[90,2] + -10.332;
   1:  PR[91,3] = PR[90,3] + 101.683;
   1:L PR[91] R[100]mm/sec CNT100;
   1:  PR[91,1] = PR[90,1] + -39.085;
   1:  PR[91,2] = PR[90,2] + -12.040;
   1:  PR[91,3] = PR[90,3] + 101.694;
   1:L PR[91] R[100]mm/sec CNT100;
   1:  PR[91,1] = PR[90,1] + -39.044;
   1:  PR[91,2] = PR[90,2] + -12.076;
   1:  PR[91,3] = PR[90,3] + 101.705;
   1:L PR[91] R[100]mm/sec CNT100;
   1:  PR[91,1] = PR[90,1] + -34.789;
   1:  PR[91,2] = PR[90,2] + -15.746;
   1:L PR[91] R[100]mm/sec CNT100;
   1:  PR[91,1] = PR[90,1] + -29.226;
   1:  PR[91,2] = PR[90,2] + -19.263;
   1:  PR[91,3] = PR[90,3] + 101.732;
   1:L PR[91] R[100]mm/sec CNT100;
   1:  PR[91,1] = PR[90,1] + -22.441;
   1:  PR[91,2] = PR[90,2] + -22.483;
   1:  PR[91,3] = PR[90,3] + 101.763;
   1:L PR[91] R[100]mm/sec CNT100;
   1:  PR[91,1] = PR[90,1] + -14.522;
   1:  PR[91,2] = PR[90,2] + -25.319;
   1:  PR[91,3] = PR[90,3] + 101.799;
   1:L PR[91] R[100]mm/sec CNT100;
   1:  PR[91,1] = PR[90,1] + -5.574;
   1:  PR[91,2] = PR[90,2] + -27.678;
   1:  PR[91,3] = PR[90,3] + 101.839;
   1:L PR[91] R[100]mm/sec CNT100;
   1:  PR[91,1] = PR[90,1] + 3.318;
   1:  PR[91,2] = PR[90,2] + -29.304;
   1:  PR[91,3] = PR[90,3] + 101.883;
   1:L PR[91] R[100]mm/sec CNT100;
   1:  PR[91,1] = PR[90,1] + 3.961;
   1:  PR[91,2] = PR[90,2] + -29.449;
   1:  PR[91,3] = PR[90,3] + 101.926;
   1:L PR[91] R[100]mm/sec CNT100;
   1:  PR[91,1] = PR[90,1] + 5.231;
   1:  PR[91,2] = PR[90,2] + -29.640;
   1:  PR[91,3] = PR[90,3] + 101.929;
   1:L PR[91] R[100]mm/sec CNT100;
   1:  PR[91,1] = PR[90,1] + 11.669;
   1:  PR[91,2] = PR[90,2] + -30.517;
   1:  PR[91,3] = PR[90,3] + 101.935;
   1:L PR[91] R[100]mm/sec CNT100;
   1:  PR[91,1] = PR[90,1] + 16.200;
   1:  PR[91,2] = PR[90,2] + -30.758;
   1:  PR[91,3] = PR[90,3] + 101.966;
   1:L PR[91] R[100]mm/sec CNT100;
   1:  PR[91,1] = PR[90,1] + 21.247;
   1:  PR[91,2] = PR[90,2] + -31.088;
   1:  PR[91,3] = PR[90,3] + 101.987;
   1:L PR[91] R[100]mm/sec CNT100;
   1:  PR[91,1] = PR[90,1] + 21.711;
   1:  PR[91,2] = PR[90,2] + -31.096;
   1:  PR[91,3] = PR[90,3] + 102.011;
   1:L PR[91] R[100]mm/sec CNT100;
   1:  PR[91,1] = PR[90,1] + 27.454;
   1:  PR[91,2] = PR[90,2] + -30.791;
   1:  PR[91,3] = PR[90,3] + 102.014;
   1:L PR[91] R[100]mm/sec CNT100;
   1:  PR[91,1] = PR[90,1] + 27.282;
   1:  PR[91,2] = PR[90,2] + -31.403;
   1:  PR[91,3] = PR[90,3] + 102.041;
   1:L PR[91] R[100]mm/sec CNT100;
   1:  PR[91,1] = PR[90,1] + 27.911;
   1:  PR[91,2] = PR[90,2] + -31.505;
   1:  PR[91,3] = PR[90,3] + 102.044;
   1:L PR[91] R[100]mm/sec CNT100;
   1:  PR[91,1] = PR[90,1] + 28.439;
   1:  PR[91,2] = PR[90,2] + -31.566;
   1:  PR[91,3] = PR[90,3] + 102.047;
   1:L PR[91] R[100]mm/sec CNT100;
   1:  PR[91,1] = PR[90,1] + 30.355;
   1:  PR[91,2] = PR[90,2] + -31.693;
   1:  PR[91,3] = PR[90,3] + 102.050;
   1:L PR[91] R[100]mm/sec CNT100;
   1:  PR[91,1] = PR[90,1] + 33.991;
   1:  PR[91,2] = PR[90,2] + -31.618;
   1:  PR[91,3] = PR[90,3] + 102.059;
   1:L PR[91] R[100]mm/sec CNT100;
   1:  PR[91,1] = PR[90,1] + 35.961;
   1:  PR[91,2] = PR[90,2] + -31.416;
   1:  PR[91,3] = PR[90,3] + 102.076;
   1:L PR[91] R[100]mm/sec CNT100;
   1:  PR[91,1] = PR[90,1] + 39.430;
   1:  PR[91,2] = PR[90,2] + -30.690;
   1:  PR[91,3] = PR[90,3] + 102.085;
   1:L PR[91] R[100]mm/sec CNT100;
   1:  PR[91,1] = PR[90,1] + 41.418;
   1:  PR[91,2] = PR[90,2] + -30.135;
   1:  PR[91,3] = PR[90,3] + 102.102;
   1:L PR[91] R[100]mm/sec CNT100;
   1:  PR[91,1] = PR[90,1] + 44.584;
   1:  PR[91,2] = PR[90,2] + -28.830;
   1:  PR[91,3] = PR[90,3] + 102.112;
   1:L PR[91] R[100]mm/sec CNT100;
   1:  PR[91,1] = PR[90,1] + 46.547;
   1:  PR[91,2] = PR[90,2] + -27.900;
   1:  PR[91,3] = PR[90,3] + 102.128;
   1:L PR[91] R[100]mm/sec CNT100;
   1:  PR[91,1] = PR[90,1] + 49.293;
   1:  PR[91,2] = PR[90,2] + -26.117;
   1:  PR[91,3] = PR[90,3] + 102.139;
   1:L PR[91] R[100]mm/sec CNT100;
   1:  PR[91,1] = PR[90,1] + 51.187;
   1:  PR[91,2] = PR[90,2] + -24.788;
   1:  PR[91,3] = PR[90,3] + 102.154;
   1:L PR[91] R[100]mm/sec CNT100;
   1:  PR[91,1] = PR[90,1] + 53.422;
   1:  PR[91,2] = PR[90,2] + -22.669;
   1:  PR[91,3] = PR[90,3] + 102.165;
   1:L PR[91] R[100]mm/sec CNT100;
   1:  PR[91,1] = PR[90,1] + 55.187;
   1:  PR[91,2] = PR[90,2] + -20.915;
   1:  PR[91,3] = PR[90,3] + 102.180;
   1:L PR[91] R[100]mm/sec CNT100;
   1:  PR[91,1] = PR[90,1] + 56.859;
   1:  PR[91,2] = PR[90,2] + -18.617;
   1:  PR[91,3] = PR[90,3] + 102.192;
   1:L PR[91] R[100]mm/sec CNT100;
   1:  PR[91,1] = PR[90,1] + 58.424;
   1:  PR[91,2] = PR[90,2] + -16.414;
   1:  PR[91,3] = PR[90,3] + 102.205;
   1:L PR[91] R[100]mm/sec CNT100;
   1:  PR[91,1] = PR[90,1] + 60.806;
   1:  PR[91,2] = PR[90,2] + -11.438;
   1:  PR[91,3] = PR[90,3] + 102.218;
   1:L PR[91] R[100]mm/sec CNT100;
   1:  PR[91,1] = PR[90,1] + 62.257;
   1:  PR[91,2] = PR[90,2] + -6.156;
   1:  PR[91,3] = PR[90,3] + 102.244;
   1:L PR[91] R[100]mm/sec CNT100;
   1:  PR[91,1] = PR[90,1] + 62.750;
   1:  PR[91,2] = PR[90,2] + -0.729;
   1:  PR[91,3] = PR[90,3] + 102.271;
   1:L PR[91] R[100]mm/sec CNT100;
   1:  PR[91,1] = PR[90,1] + 62.257;
   1:  PR[91,2] = PR[90,2] + 4.698;
   1:  PR[91,3] = PR[90,3] + 102.296;
   1:L PR[91] R[100]mm/sec CNT100;
   1:  PR[91,1] = PR[90,1] + 60.805;
   1:  PR[91,2] = PR[90,2] + 9.981;
   1:  PR[91,3] = PR[90,3] + 102.322;
   1:L PR[91] R[100]mm/sec CNT100;
   1:  PR[91,1] = PR[90,1] + 58.423;
   1:  PR[91,2] = PR[90,2] + 14.957;
   1:  PR[91,3] = PR[90,3] + 102.348;
   1:L PR[91] R[100]mm/sec CNT100;
   1:  PR[91,1] = PR[90,1] + 56.858;
   1:  PR[91,2] = PR[90,2] + 17.160;
   1:  PR[91,3] = PR[90,3] + 102.375;
   1:L PR[91] R[100]mm/sec CNT100;
   1:  PR[91,1] = PR[90,1] + 55.186;
   1:  PR[91,2] = PR[90,2] + 19.458;
   1:  PR[91,3] = PR[90,3] + 102.388;
   1:L PR[91] R[100]mm/sec CNT100;
   1:  PR[91,1] = PR[90,1] + 53.420;
   1:  PR[91,2] = PR[90,2] + 21.211;
   1:  PR[91,3] = PR[90,3] + 102.401;
   1:L PR[91] R[100]mm/sec CNT100;
   1:  PR[91,1] = PR[90,1] + 51.185;
   1:  PR[91,2] = PR[90,2] + 23.331;
   1:  PR[91,3] = PR[90,3] + 102.413;
   1:L PR[91] R[100]mm/sec CNT100;
   1:  PR[91,1] = PR[90,1] + 49.292;
   1:  PR[91,2] = PR[90,2] + 24.658;
   1:  PR[91,3] = PR[90,3] + 102.428;
   1:L PR[91] R[100]mm/sec CNT100;
   1:  PR[91,1] = PR[90,1] + 46.545;
   1:  PR[91,2] = PR[90,2] + 26.442;
   1:  PR[91,3] = PR[90,3] + 102.439;
   1:L PR[91] R[100]mm/sec CNT100;
   1:  PR[91,1] = PR[90,1] + 44.583;
   1:  PR[91,2] = PR[90,2] + 27.370;
   1:  PR[91,3] = PR[90,3] + 102.454;
   1:L PR[91] R[100]mm/sec CNT100;
   1:  PR[91,1] = PR[90,1] + 41.417;
   1:  PR[91,2] = PR[90,2] + 28.677;
   1:  PR[91,3] = PR[90,3] + 102.464;
   1:L PR[91] R[100]mm/sec CNT100;
   1:  PR[91,1] = PR[90,1] + 39.430;
   1:  PR[91,2] = PR[90,2] + 29.230;
   1:  PR[91,3] = PR[90,3] + 102.481;
   1:L PR[91] R[100]mm/sec CNT100;
   1:  PR[91,1] = PR[90,1] + 35.960;
   1:  PR[91,2] = PR[90,2] + 29.958;
   1:  PR[91,3] = PR[90,3] + 102.491;
   1:L PR[91] R[100]mm/sec CNT100;
   1:  PR[91,1] = PR[90,1] + 33.991;
   1:  PR[91,2] = PR[90,2] + 30.159;
   1:  PR[91,3] = PR[90,3] + 102.507;
   1:L PR[91] R[100]mm/sec CNT100;
   1:  PR[91,1] = PR[90,1] + 30.354;
   1:  PR[91,2] = PR[90,2] + 30.234;
   1:  PR[91,3] = PR[90,3] + 102.517;
   1:L PR[91] R[100]mm/sec CNT100;
   1:  PR[91,1] = PR[90,1] + 28.440;
   1:  PR[91,2] = PR[90,2] + 30.107;
   1:  PR[91,3] = PR[90,3] + 102.534;
   1:L PR[91] R[100]mm/sec CNT100;
   1:  PR[91,1] = PR[90,1] + 27.822;
   1:  PR[91,2] = PR[90,2] + 30.035;
   1:  PR[91,3] = PR[90,3] + 102.543;
   1:L PR[91] R[100]mm/sec CNT100;
   1:  PR[91,1] = PR[90,1] + 24.884;
   1:  PR[91,2] = PR[90,2] + 29.559;
   1:  PR[91,3] = PR[90,3] + 102.546;
   1:L PR[91] R[100]mm/sec CNT100;
   1:  PR[91,1] = PR[90,1] + 21.832;
   1:  PR[91,2] = PR[90,2] + 29.638;
   1:  PR[91,3] = PR[90,3] + 102.560;
   1:L PR[91] R[100]mm/sec CNT100;
   1:  PR[91,1] = PR[90,1] + 21.252;
   1:  PR[91,2] = PR[90,2] + 29.629;
   1:  PR[91,3] = PR[90,3] + 102.575;
   1:L PR[91] R[100]mm/sec CNT100;
   1:  PR[91,1] = PR[90,1] + 16.200;
   1:  PR[91,2] = PR[90,2] + 29.300;
   1:  PR[91,3] = PR[90,3] + 102.578;
   1:L PR[91] R[100]mm/sec CNT100;
   1:  PR[91,1] = PR[90,1] + 11.670;
   1:  PR[91,2] = PR[90,2] + 29.058;
   1:  PR[91,3] = PR[90,3] + 102.602;
   1:L PR[91] R[100]mm/sec CNT100;
   1:  PR[91,1] = PR[90,1] + 5.231;
   1:  PR[91,2] = PR[90,2] + 28.182;
   1:  PR[91,3] = PR[90,3] + 102.623;
   1:L PR[91] R[100]mm/sec CNT100;
   1:  PR[91,1] = PR[90,1] + 3.961;
   1:  PR[91,2] = PR[90,2] + 27.990;
   1:  PR[91,3] = PR[90,3] + 102.654;
   1:L PR[91] R[100]mm/sec CNT100;
   1:  PR[91,1] = PR[90,1] + 3.318;
   1:  PR[91,2] = PR[90,2] + 27.846;
   1:  PR[91,3] = PR[90,3] + 102.660;
   1:L PR[91] R[100]mm/sec CNT100;
   1:  PR[91,1] = PR[90,1] + -5.574;
   1:  PR[91,2] = PR[90,2] + 26.220;
   1:  PR[91,3] = PR[90,3] + 102.664;
   1:L PR[91] R[100]mm/sec CNT100;
   1:  PR[91,1] = PR[90,1] + -14.522;
   1:  PR[91,2] = PR[90,2] + 23.860;
   1:  PR[91,3] = PR[90,3] + 102.707;
   1:L PR[91] R[100]mm/sec CNT100;
   1:  PR[91,1] = PR[90,1] + -22.442;
   1:  PR[91,2] = PR[90,2] + 21.024;
   1:  PR[91,3] = PR[90,3] + 102.751;
   1:L PR[91] R[100]mm/sec CNT100;
   1:  PR[91,1] = PR[90,1] + -27.000;
   1:  PR[91,2] = PR[90,2] + 18.869;
   1:  PR[91,3] = PR[90,3] + 102.791;
   1:L PR[91] R[100]mm/sec CNT100;
   1:  PR[91,1] = PR[90,1] + -29.223;
   1:  PR[91,2] = PR[90,2] + 17.806;
   1:  PR[91,3] = PR[90,3] + 102.815;
   1:L PR[91] R[100]mm/sec CNT100;
   1:  PR[91,1] = PR[90,1] + -34.789;
   1:  PR[91,2] = PR[90,2] + 14.288;
   1:  PR[91,3] = PR[90,3] + 102.826;
   1:L PR[91] R[100]mm/sec CNT100;
   1:  PR[91,1] = PR[90,1] + -39.088;
   1:  PR[91,2] = PR[90,2] + 10.578;
   1:  PR[91,3] = PR[90,3] + 102.858;
   1:L PR[91] R[100]mm/sec CNT100;
   1:  PR[91,1] = PR[90,1] + -40.442;
   1:  PR[91,2] = PR[90,2] + 8.868;
   1:  PR[91,3] = PR[90,3] + 102.885;
   1:L PR[91] R[100]mm/sec CNT100;
   1:  PR[91] = PR[90];
   1:  PR[91,1] = PR[90,1] + -40.854;
   1:  PR[91,2] = PR[90,2] + 4.880;
   1:  PR[91,3] = PR[90,3] + 104.195;
   1:L PR[91] R[100]mm/sec CNT100;
   1:  PR[91,1] = PR[90,1] + -41.599;
   1:  PR[91,2] = PR[90,2] + 3.126;
   1:  PR[91,3] = PR[90,3] + 102.905;
   1:L PR[91] R[100]mm/sec CNT100;
   1:  PR[91,1] = PR[90,1] + -41.622;
   1:  PR[91,2] = PR[90,2] + 3.002;
   1:  PR[91,3] = PR[90,3] + 102.915;
   1:L PR[91] R[100]mm/sec CNT100;
   1:  PR[91,1] = PR[90,1] + -42.130;
   1:  PR[91,2] = PR[90,2] + -0.655;
   1:L PR[91] R[100]mm/sec CNT100;
   1:  PR[91,1] = PR[90,1] + -42.075;
   1:  PR[91,2] = PR[90,2] + -0.913;
   1:  PR[91,3] = PR[90,3] + 102.933;
   1:L PR[91] R[100]mm/sec CNT100;
   1:  PR[91,1] = PR[90,1] + -41.574;
   1:  PR[91,2] = PR[90,2] + -4.626;
   1:  PR[91,3] = PR[90,3] + 102.934;
   1:L PR[91] R[100]mm/sec CNT100;
   1:  PR[91,1] = PR[90,1] + -40.853;
   1:  PR[91,2] = PR[90,2] + -6.342;
   1:  PR[91,3] = PR[90,3] + 102.952;
   1:L PR[91] R[100]mm/sec CNT100;
   1:  PR[91,1] = PR[90,1] + -39.945;
   1:  PR[91,2] = PR[90,2] + -8.308;
   1:  PR[91,3] = PR[90,3] + 102.961;
   1:L PR[91] R[100]mm/sec CNT100;
   1:  PR[91,1] = PR[90,1] + -36.918;
   1:  PR[91,2] = PR[90,2] + -12.128;
   1:  PR[91,3] = PR[90,3] + 102.972;
   1:L PR[91] R[100]mm/sec CNT100;
   1:  PR[91,1] = PR[90,1] + -32.589;
   1:  PR[91,2] = PR[90,2] + -15.867;
   1:  PR[91,3] = PR[90,3] + 102.995;
   1:L PR[91] R[100]mm/sec CNT100;
   1:  PR[91,1] = PR[90,1] + -26.988;
   1:  PR[91,2] = PR[90,2] + -19.410;
   1:  PR[91,3] = PR[90,3] + 103.022;
   1:L PR[91] R[100]mm/sec CNT100;
   1:  PR[91,1] = PR[90,1] + -20.156;
   1:  PR[91,2] = PR[90,2] + -22.656;
   1:  PR[91,3] = PR[90,3] + 103.054;
   1:L PR[91] R[100]mm/sec CNT100;
   1:  PR[91,1] = PR[90,1] + -12.183;
   1:  PR[91,2] = PR[90,2] + -25.515;
   1:  PR[91,3] = PR[90,3] + 103.091;
   1:L PR[91] R[100]mm/sec CNT100;
   1:  PR[91,1] = PR[90,1] + -3.172;
   1:  PR[91,2] = PR[90,2] + -27.894;
   1:  PR[91,3] = PR[90,3] + 103.131;
   1:L PR[91] R[100]mm/sec CNT100;
   1:  PR[91,1] = PR[90,1] + 2.669;
   1:  PR[91,2] = PR[90,2] + -28.962;
   1:  PR[91,3] = PR[90,3] + 103.176;
   1:L PR[91] R[100]mm/sec CNT100;
   1:  PR[91,1] = PR[90,1] + 5.288;
   1:  PR[91,2] = PR[90,2] + -29.551;
   1:  PR[91,3] = PR[90,3] + 103.204;
   1:L PR[91] R[100]mm/sec CNT100;
   1:  PR[91,1] = PR[90,1] + 10.524;
   1:  PR[91,2] = PR[90,2] + -30.341;
   1:  PR[91,3] = PR[90,3] + 103.217;
   1:L PR[91] R[100]mm/sec CNT100;
   1:  PR[91,1] = PR[90,1] + 13.345;
   1:  PR[91,2] = PR[90,2] + -30.725;
   1:  PR[91,3] = PR[90,3] + 103.243;
   1:L PR[91] R[100]mm/sec CNT100;
   1:  PR[91,1] = PR[90,1] + 15.328;
   1:  PR[91,2] = PR[90,2] + -30.830;
   1:  PR[91,3] = PR[90,3] + 103.256;
   1:L PR[91] R[100]mm/sec CNT100;
   1:  PR[91,1] = PR[90,1] + 22.782;
   1:  PR[91,2] = PR[90,2] + -31.317;
   1:  PR[91,3] = PR[90,3] + 103.266;
   1:L PR[91] R[100]mm/sec CNT100;
   1:  PR[91,1] = PR[90,1] + 23.522;
   1:  PR[91,2] = PR[90,2] + -31.330;
   1:  PR[91,3] = PR[90,3] + 103.302;
   1:L PR[91] R[100]mm/sec CNT100;
   1:  PR[91,1] = PR[90,1] + 28.057;
   1:  PR[91,2] = PR[90,2] + -31.089;
   1:  PR[91,3] = PR[90,3] + 103.305;
   1:L PR[91] R[100]mm/sec CNT100;
   1:  PR[91,1] = PR[90,1] + 27.901;
   1:  PR[91,2] = PR[90,2] + -31.644;
   1:  PR[91,3] = PR[90,3] + 103.327;
   1:L PR[91] R[100]mm/sec CNT100;
   1:  PR[91,1] = PR[90,1] + 28.182;
   1:  PR[91,2] = PR[90,2] + -31.677;
   1:  PR[91,3] = PR[90,3] + 103.330;
   1:L PR[91] R[100]mm/sec CNT100;
   1:  PR[91,1] = PR[90,1] + 31.039;
   1:  PR[91,2] = PR[90,2] + -31.866;
   1:  PR[91,3] = PR[90,3] + 103.331;
   1:L PR[91] R[100]mm/sec CNT100;
   1:  PR[91,1] = PR[90,1] + 33.625;
   1:  PR[91,2] = PR[90,2] + -31.813;
   1:  PR[91,3] = PR[90,3] + 103.345;
   1:L PR[91] R[100]mm/sec CNT100;
   1:  PR[91,1] = PR[90,1] + 36.676;
   1:  PR[91,2] = PR[90,2] + -31.499;
   1:  PR[91,3] = PR[90,3] + 103.358;
   1:L PR[91] R[100]mm/sec CNT100;
   1:  PR[91,1] = PR[90,1] + 38.974;
   1:  PR[91,2] = PR[90,2] + -31.019;
   1:  PR[91,3] = PR[90,3] + 103.372;
   1:L PR[91] R[100]mm/sec CNT100;
   1:  PR[91,1] = PR[90,1] + 42.154;
   1:  PR[91,2] = PR[90,2] + -30.132;
   1:  PR[91,3] = PR[90,3] + 103.384;
   1:L PR[91] R[100]mm/sec CNT100;
   1:  PR[91,1] = PR[90,1] + 44.040;
   1:  PR[91,2] = PR[90,2] + -29.354;
   1:  PR[91,3] = PR[90,3] + 103.399;
   1:L PR[91] R[100]mm/sec CNT100;
   1:  PR[91,1] = PR[90,1] + 47.292;
   1:  PR[91,2] = PR[90,2] + -27.813;
   1:  PR[91,3] = PR[90,3] + 103.409;
   1:L PR[91] R[100]mm/sec CNT100;
   1:  PR[91,1] = PR[90,1] + 48.678;
   1:  PR[91,2] = PR[90,2] + -26.913;
   1:  PR[91,3] = PR[90,3] + 103.426;
   1:L PR[91] R[100]mm/sec CNT100;
   1:  PR[91,1] = PR[90,1] + 51.932;
   1:  PR[91,2] = PR[90,2] + -24.631;
   1:  PR[91,3] = PR[90,3] + 103.434;
   1:L PR[91] R[100]mm/sec CNT100;
   1:  PR[91,1] = PR[90,1] + 52.776;
   1:  PR[91,2] = PR[90,2] + -23.830;
   1:  PR[91,3] = PR[90,3] + 103.454;
   1:L PR[91] R[100]mm/sec CNT100;
   1:  PR[91,1] = PR[90,1] + 55.913;
   1:  PR[91,2] = PR[90,2] + -20.714;
   1:  PR[91,3] = PR[90,3] + 103.459;
   1:L PR[91] R[100]mm/sec CNT100;
   1:  PR[91,1] = PR[90,1] + 59.142;
   1:  PR[91,2] = PR[90,2] + -16.184;
   1:  PR[91,3] = PR[90,3] + 103.480;
   1:L PR[91] R[100]mm/sec CNT100;
   1:  PR[91,1] = PR[90,1] + 61.491;
   1:  PR[91,2] = PR[90,2] + -11.347;
   1:  PR[91,3] = PR[90,3] + 103.507;
   1:L PR[91] R[100]mm/sec CNT100;
   1:  PR[91,1] = PR[90,1] + 61.672;
   1:  PR[91,2] = PR[90,2] + -10.773;
   1:  PR[91,3] = PR[90,3] + 103.533;
   1:L PR[91] R[100]mm/sec CNT100;
   1:  PR[91,1] = PR[90,1] + 62.960;
   1:  PR[91,2] = PR[90,2] + -6.180;
   1:  PR[91,3] = PR[90,3] + 103.536;
   1:L PR[91] R[100]mm/sec CNT100;
   1:  PR[91,1] = PR[90,1] + 63.465;
   1:  PR[91,2] = PR[90,2] + -0.726;
   1:  PR[91,3] = PR[90,3] + 103.559;
   1:L PR[91] R[100]mm/sec CNT100;
   1:  PR[91,1] = PR[90,1] + 63.094;
   1:  PR[91,2] = PR[90,2] + 3.412;
   1:  PR[91,3] = PR[90,3] + 103.585;
   1:L PR[91] R[100]mm/sec CNT100;
   1:  PR[91,1] = PR[90,1] + 62.962;
   1:  PR[91,2] = PR[90,2] + 4.714;
   1:  PR[91,3] = PR[90,3] + 103.605;
   1:L PR[91] R[100]mm/sec CNT100;
   1:  PR[91,1] = PR[90,1] + 61.670;
   1:  PR[91,2] = PR[90,2] + 9.319;
   1:  PR[91,3] = PR[90,3] + 103.611;
   1:L PR[91] R[100]mm/sec CNT100;
   1:  PR[91,1] = PR[90,1] + 61.489;
   1:  PR[91,2] = PR[90,2] + 9.892;
   1:  PR[91,3] = PR[90,3] + 103.634;
   1:L PR[91] R[100]mm/sec CNT100;
   1:  PR[91,1] = PR[90,1] + 59.138;
   1:  PR[91,2] = PR[90,2] + 14.731;
   1:  PR[91,3] = PR[90,3] + 103.637;
   1:L PR[91] R[100]mm/sec CNT100;
   1:  PR[91,1] = PR[90,1] + 55.908;
   1:  PR[91,2] = PR[90,2] + 19.261;
   1:  PR[91,3] = PR[90,3] + 103.663;
   1:L PR[91] R[100]mm/sec CNT100;
   1:  PR[91,1] = PR[90,1] + 52.770;
   1:  PR[91,2] = PR[90,2] + 22.376;
   1:  PR[91,3] = PR[90,3] + 103.690;
   1:L PR[91] R[100]mm/sec CNT100;
   1:  PR[91,1] = PR[90,1] + 51.925;
   1:  PR[91,2] = PR[90,2] + 23.177;
   1:  PR[91,3] = PR[90,3] + 103.711;
   1:L PR[91] R[100]mm/sec CNT100;
   1:  PR[91,1] = PR[90,1] + 48.672;
   1:  PR[91,2] = PR[90,2] + 25.458;
   1:  PR[91,3] = PR[90,3] + 103.716;
   1:L PR[91] R[100]mm/sec CNT100;
   1:  PR[91,1] = PR[90,1] + 47.285;
   1:  PR[91,2] = PR[90,2] + 26.358;
   1:  PR[91,3] = PR[90,3] + 103.736;
   1:L PR[91] R[100]mm/sec CNT100;
   1:  PR[91,1] = PR[90,1] + 44.034;
   1:  PR[91,2] = PR[90,2] + 27.897;
   1:  PR[91,3] = PR[90,3] + 103.743;
   1:L PR[91] R[100]mm/sec CNT100;
   1:  PR[91,1] = PR[90,1] + 42.147;
   1:  PR[91,2] = PR[90,2] + 28.676;
   1:  PR[91,3] = PR[90,3] + 103.761;
   1:L PR[91] R[100]mm/sec CNT100;
   1:  PR[91,1] = PR[90,1] + 38.968;
   1:  PR[91,2] = PR[90,2] + 29.560;
   1:  PR[91,3] = PR[90,3] + 103.771;
   1:L PR[91] R[100]mm/sec CNT100;
   1:  PR[91,1] = PR[90,1] + 36.669;
   1:  PR[91,2] = PR[90,2] + 30.042;
   1:  PR[91,3] = PR[90,3] + 103.786;
   1:L PR[91] R[100]mm/sec CNT100;
   1:  PR[91,1] = PR[90,1] + 33.620;
   1:  PR[91,2] = PR[90,2] + 30.354;
   1:  PR[91,3] = PR[90,3] + 103.798;
   1:L PR[91] R[100]mm/sec CNT100;
   1:  PR[91,1] = PR[90,1] + 31.032;
   1:  PR[91,2] = PR[90,2] + 30.407;
   1:  PR[91,3] = PR[90,3] + 103.812;
   1:L PR[91] R[100]mm/sec CNT100;
   1:  PR[91,1] = PR[90,1] + 28.177;
   1:  PR[91,2] = PR[90,2] + 30.217;
   1:  PR[91,3] = PR[90,3] + 103.825;
   1:L PR[91] R[100]mm/sec CNT100;
   1:  PR[91,1] = PR[90,1] + 27.233;
   1:  PR[91,2] = PR[90,2] + 30.107;
   1:  PR[91,3] = PR[90,3] + 103.839;
   1:L PR[91] R[100]mm/sec CNT100;
   1:  PR[91,1] = PR[90,1] + 25.494;
   1:  PR[91,2] = PR[90,2] + 29.826;
   1:  PR[91,3] = PR[90,3] + 103.843;
   1:L PR[91] R[100]mm/sec CNT100;
   1:  PR[91,1] = PR[90,1] + 23.688;
   1:  PR[91,2] = PR[90,2] + 29.873;
   1:  PR[91,3] = PR[90,3] + 103.852;
   1:L PR[91] R[100]mm/sec CNT100;
   1:  PR[91,1] = PR[90,1] + 22.790;
   1:  PR[91,2] = PR[90,2] + 29.858;
   1:  PR[91,3] = PR[90,3] + 103.860;
   1:L PR[91] R[100]mm/sec CNT100;
   1:  PR[91,1] = PR[90,1] + 15.328;
   1:  PR[91,2] = PR[90,2] + 29.372;
   1:  PR[91,3] = PR[90,3] + 103.865;
   1:L PR[91] R[100]mm/sec CNT100;
   1:  PR[91,1] = PR[90,1] + 13.346;
   1:  PR[91,2] = PR[90,2] + 29.266;
   1:  PR[91,3] = PR[90,3] + 103.900;
   1:L PR[91] R[100]mm/sec CNT100;
   1:  PR[91,1] = PR[90,1] + 10.526;
   1:  PR[91,2] = PR[90,2] + 28.882;
   1:  PR[91,3] = PR[90,3] + 103.910;
   1:L PR[91] R[100]mm/sec CNT100;
   1:  PR[91,1] = PR[90,1] + 5.288;
   1:  PR[91,2] = PR[90,2] + 28.093;
   1:  PR[91,3] = PR[90,3] + 103.924;
   1:L PR[91] R[100]mm/sec CNT100;
   1:  PR[91,1] = PR[90,1] + 2.669;
   1:  PR[91,2] = PR[90,2] + 27.503;
   1:  PR[91,3] = PR[90,3] + 103.949;
   1:L PR[91] R[100]mm/sec CNT100;
   1:  PR[91,1] = PR[90,1] + -3.172;
   1:  PR[91,2] = PR[90,2] + 26.435;
   1:  PR[91,3] = PR[90,3] + 103.962;
   1:L PR[91] R[100]mm/sec CNT100;
   1:  PR[91,1] = PR[90,1] + -12.183;
   1:  PR[91,2] = PR[90,2] + 24.056;
   1:  PR[91,3] = PR[90,3] + 103.991;
   1:L PR[91] R[100]mm/sec CNT100;
   1:  PR[91,1] = PR[90,1] + -20.156;
   1:  PR[91,2] = PR[90,2] + 21.198;
   1:  PR[91,3] = PR[90,3] + 104.035;
   1:L PR[91] R[100]mm/sec CNT100;
   1:  PR[91,1] = PR[90,1] + -26.988;
   1:  PR[91,2] = PR[90,2] + 17.952;
   1:  PR[91,3] = PR[90,3] + 104.076;
   1:L PR[91] R[100]mm/sec CNT100;
   1:  PR[91,1] = PR[90,1] + -32.589;
   1:  PR[91,2] = PR[90,2] + 14.408;
   1:  PR[91,3] = PR[90,3] + 104.112;
   1:L PR[91] R[100]mm/sec CNT100;
   1:  PR[91,1] = PR[90,1] + -36.918;
   1:  PR[91,2] = PR[90,2] + 10.669;
   1:  PR[91,3] = PR[90,3] + 104.144;
   1:L PR[91] R[100]mm/sec CNT100;
   1:  PR[91,1] = PR[90,1] + -39.945;
   1:  PR[91,2] = PR[90,2] + 6.849;
   1:  PR[91,3] = PR[90,3] + 104.172;
   1:L PR[91] R[100]mm/sec CNT100;
   1:  PR[91] = PR[90];
   1:  PR[91,1] = PR[90,1] + -39.573;
   1:  PR[91,2] = PR[90,2] + 3.064;
   1:  PR[91,3] = PR[90,3] + 105.495;
   1:L PR[91] R[100]mm/sec CNT100;
   1:  PR[91,1] = PR[90,1] + -40.152;
   1:  PR[91,2] = PR[90,2] + -0.729;
   1:  PR[91,3] = PR[90,3] + 104.216;
   1:L PR[91] R[100]mm/sec CNT100;
   1:  PR[91,1] = PR[90,1] + -39.573;
   1:  PR[91,2] = PR[90,2] + -4.523;
   1:  PR[91,3] = PR[90,3] + 104.234;
   1:L PR[91] R[100]mm/sec CNT100;
   1:  PR[91,1] = PR[90,1] + -37.797;
   1:  PR[91,2] = PR[90,2] + -8.370;
   1:  PR[91,3] = PR[90,3] + 104.253;
   1:L PR[91] R[100]mm/sec CNT100;
   1:  PR[91,1] = PR[90,1] + -34.746;
   1:  PR[91,2] = PR[90,2] + -12.223;
   1:  PR[91,3] = PR[90,3] + 104.273;
   1:L PR[91] R[100]mm/sec CNT100;
   1:  PR[91,1] = PR[90,1] + -34.005;
   1:  PR[91,2] = PR[90,2] + -12.868;
   1:  PR[91,3] = PR[90,3] + 104.297;
   1:L PR[91] R[100]mm/sec CNT100;
   1:  PR[91,1] = PR[90,1] + -30.390;
   1:  PR[91,2] = PR[90,2] + -15.987;
   1:  PR[91,3] = PR[90,3] + 104.302;
   1:L PR[91] R[100]mm/sec CNT100;
   1:  PR[91,1] = PR[90,1] + -24.750;
   1:  PR[91,2] = PR[90,2] + -19.558;
   1:  PR[91,3] = PR[90,3] + 104.325;
   1:L PR[91] R[100]mm/sec CNT100;
   1:  PR[91,1] = PR[90,1] + -17.871;
   1:  PR[91,2] = PR[90,2] + -22.829;
   1:  PR[91,3] = PR[90,3] + 104.357;
   1:L PR[91] R[100]mm/sec CNT100;
   1:  PR[91,1] = PR[90,1] + -9.843;
   1:  PR[91,2] = PR[90,2] + -25.710;
   1:  PR[91,3] = PR[90,3] + 104.394;
   1:L PR[91] R[100]mm/sec CNT100;
   1:  PR[91,1] = PR[90,1] + -0.771;
   1:  PR[91,2] = PR[90,2] + -28.110;
   1:  PR[91,3] = PR[90,3] + 104.436;
   1:L PR[91] R[100]mm/sec CNT100;
   1:  PR[91,1] = PR[90,1] + 2.021;
   1:  PR[91,2] = PR[90,2] + -28.620;
   1:  PR[91,3] = PR[90,3] + 104.481;
   1:L PR[91] R[100]mm/sec CNT100;
   1:  PR[91,1] = PR[90,1] + 6.614;
   1:  PR[91,2] = PR[90,2] + -29.654;
   1:  PR[91,3] = PR[90,3] + 104.495;
   1:L PR[91] R[100]mm/sec CNT100;
   1:  PR[91,1] = PR[90,1] + 14.674;
   1:  PR[91,2] = PR[90,2] + -30.869;
   1:  PR[91,3] = PR[90,3] + 104.518;
   1:L PR[91] R[100]mm/sec CNT100;
   1:  PR[91,1] = PR[90,1] + 15.053;
   1:  PR[91,2] = PR[90,2] + -30.940;
   1:  PR[91,3] = PR[90,3] + 104.557;
   1:L PR[91] R[100]mm/sec CNT100;
   1:  PR[91,1] = PR[90,1] + 24.318;
   1:  PR[91,2] = PR[90,2] + -31.546;
   1:  PR[91,3] = PR[90,3] + 104.559;
   1:L PR[91] R[100]mm/sec CNT100;
   1:  PR[91,1] = PR[90,1] + 25.334;
   1:  PR[91,2] = PR[90,2] + -31.564;
   1:  PR[91,3] = PR[90,3] + 104.604;
   1:L PR[91] R[100]mm/sec CNT100;
   1:  PR[91,1] = PR[90,1] + 28.659;
   1:  PR[91,2] = PR[90,2] + -31.388;
   1:  PR[91,3] = PR[90,3] + 104.609;
   1:L PR[91] R[100]mm/sec CNT100;
   1:  PR[91,1] = PR[90,1] + 28.535;
   1:  PR[91,2] = PR[90,2] + -31.828;
   1:  PR[91,3] = PR[90,3] + 104.625;
   1:L PR[91] R[100]mm/sec CNT100;
   1:  PR[91,1] = PR[90,1] + 31.723;
   1:  PR[91,2] = PR[90,2] + -32.039;
   1:  PR[91,3] = PR[90,3] + 104.627;
   1:L PR[91] R[100]mm/sec CNT100;
   1:  PR[91,1] = PR[90,1] + 33.260;
   1:  PR[91,2] = PR[90,2] + -32.007;
   1:  PR[91,3] = PR[90,3] + 104.643;
   1:L PR[91] R[100]mm/sec CNT100;
   1:  PR[91,1] = PR[90,1] + 37.391;
   1:  PR[91,2] = PR[90,2] + -31.583;
   1:  PR[91,3] = PR[90,3] + 104.650;
   1:L PR[91] R[100]mm/sec CNT100;
   1:  PR[91,1] = PR[90,1] + 38.518;
   1:  PR[91,2] = PR[90,2] + -31.347;
   1:  PR[91,3] = PR[90,3] + 104.671;
   1:L PR[91] R[100]mm/sec CNT100;
   1:  PR[91,1] = PR[90,1] + 42.890;
   1:  PR[91,2] = PR[90,2] + -30.128;
   1:  PR[91,3] = PR[90,3] + 104.676;
   1:L PR[91] R[100]mm/sec CNT100;
   1:  PR[91,1] = PR[90,1] + 43.497;
   1:  PR[91,2] = PR[90,2] + -29.878;
   1:  PR[91,3] = PR[90,3] + 104.698;
   1:L PR[91] R[100]mm/sec CNT100;
   1:  PR[91,1] = PR[90,1] + 48.014;
   1:  PR[91,2] = PR[90,2] + -27.738;
   1:  PR[91,3] = PR[90,3] + 104.701;
   1:L PR[91] R[100]mm/sec CNT100;
   1:  PR[91,1] = PR[90,1] + 52.491;
   1:  PR[91,2] = PR[90,2] + -24.657;
   1:  PR[91,3] = PR[90,3] + 104.726;
   1:L PR[91] R[100]mm/sec CNT100;
   1:  PR[91,1] = PR[90,1] + 52.939;
   1:  PR[91,2] = PR[90,2] + -24.278;
   1:  PR[91,3] = PR[90,3] + 104.752;
   1:L PR[91] R[100]mm/sec CNT100;
   1:  PR[91,1] = PR[90,1] + 56.290;
   1:  PR[91,2] = PR[90,2] + -21.026;
   1:  PR[91,3] = PR[90,3] + 104.755;
   1:L PR[91] R[100]mm/sec CNT100;
   1:  PR[91,1] = PR[90,1] + 57.496;
   1:  PR[91,2] = PR[90,2] + -19.555;
   1:  PR[91,3] = PR[90,3] + 104.777;
   1:L PR[91] R[100]mm/sec CNT100;
   1:  PR[91,1] = PR[90,1] + 59.518;
   1:  PR[91,2] = PR[90,2] + -16.773;
   1:  PR[91,3] = PR[90,3] + 104.787;
   1:L PR[91] R[100]mm/sec CNT100;
   1:  PR[91,1] = PR[90,1] + 61.164;
   1:  PR[91,2] = PR[90,2] + -13.760;
   1:  PR[91,3] = PR[90,3] + 104.803;
   1:L PR[91] R[100]mm/sec CNT100;
   1:  PR[91,1] = PR[90,1] + 62.061;
   1:  PR[91,2] = PR[90,2] + -11.918;
   1:  PR[91,3] = PR[90,3] + 104.820;
   1:L PR[91] R[100]mm/sec CNT100;
   1:  PR[91,1] = PR[90,1] + 63.499;
   1:  PR[91,2] = PR[90,2] + -7.353;
   1:  PR[91,3] = PR[90,3] + 104.830;
   1:L PR[91] R[100]mm/sec CNT100;
   1:  PR[91,1] = PR[90,1] + 63.732;
   1:  PR[91,2] = PR[90,2] + -6.522;
   1:  PR[91,3] = PR[90,3] + 104.853;
   1:L PR[91] R[100]mm/sec CNT100;
   1:  PR[91,1] = PR[90,1] + 63.816;
   1:  PR[91,2] = PR[90,2] + -5.600;
   1:  PR[91,3] = PR[90,3] + 104.857;
   1:L PR[91] R[100]mm/sec CNT100;
   1:  PR[91,1] = PR[90,1] + 64.322;
   1:  PR[91,2] = PR[90,2] + -0.727;
   1:  PR[91,3] = PR[90,3] + 104.862;
   1:L PR[91] R[100]mm/sec CNT100;
   1:  PR[91,1] = PR[90,1] + 63.735;
   1:  PR[91,2] = PR[90,2] + 5.053;
   1:  PR[91,3] = PR[90,3] + 104.886;
   1:L PR[91] R[100]mm/sec CNT100;
   1:  PR[91,1] = PR[90,1] + 63.499;
   1:  PR[91,2] = PR[90,2] + 5.895;
   1:  PR[91,3] = PR[90,3] + 104.914;
   1:L PR[91] R[100]mm/sec CNT100;
   1:  PR[91,1] = PR[90,1] + 62.061;
   1:  PR[91,2] = PR[90,2] + 10.459;
   1:  PR[91,3] = PR[90,3] + 104.918;
   1:L PR[91] R[100]mm/sec CNT100;
   1:  PR[91,1] = PR[90,1] + 61.163;
   1:  PR[91,2] = PR[90,2] + 12.302;
   1:  PR[91,3] = PR[90,3] + 104.941;
   1:L PR[91] R[100]mm/sec CNT100;
   1:  PR[91,1] = PR[90,1] + 59.516;
   1:  PR[91,2] = PR[90,2] + 15.317;
   1:  PR[91,3] = PR[90,3] + 104.951;
   1:L PR[91] R[100]mm/sec CNT100;
   1:  PR[91,1] = PR[90,1] + 57.492;
   1:  PR[91,2] = PR[90,2] + 18.101;
   1:  PR[91,3] = PR[90,3] + 104.968;
   1:L PR[91] R[100]mm/sec CNT100;
   1:  PR[91,1] = PR[90,1] + 56.286;
   1:  PR[91,2] = PR[90,2] + 19.572;
   1:  PR[91,3] = PR[90,3] + 104.984;
   1:L PR[91] R[100]mm/sec CNT100;
   1:  PR[91,1] = PR[90,1] + 52.930;
   1:  PR[91,2] = PR[90,2] + 22.827;
   1:  PR[91,3] = PR[90,3] + 104.994;
   1:L PR[91] R[100]mm/sec CNT100;
   1:  PR[91,1] = PR[90,1] + 52.482;
   1:  PR[91,2] = PR[90,2] + 23.205;
   1:  PR[91,3] = PR[90,3] + 105.016;
   1:L PR[91] R[100]mm/sec CNT100;
   1:  PR[91,1] = PR[90,1] + 48.001;
   1:  PR[91,2] = PR[90,2] + 26.286;
   1:  PR[91,3] = PR[90,3] + 105.019;
   1:L PR[91] R[100]mm/sec CNT100;
   1:  PR[91,1] = PR[90,1] + 43.484;
   1:  PR[91,2] = PR[90,2] + 28.423;
   1:  PR[91,3] = PR[90,3] + 105.046;
   1:L PR[91] R[100]mm/sec CNT100;
   1:  PR[91,1] = PR[90,1] + 42.877;
   1:  PR[91,2] = PR[90,2] + 28.674;
   1:  PR[91,3] = PR[90,3] + 105.070;
   1:L PR[91] R[100]mm/sec CNT100;
   1:  PR[91,1] = PR[90,1] + 38.506;
   1:  PR[91,2] = PR[90,2] + 29.891;
   1:  PR[91,3] = PR[90,3] + 105.073;
   1:L PR[91] R[100]mm/sec CNT100;
   1:  PR[91,1] = PR[90,1] + 37.377;
   1:  PR[91,2] = PR[90,2] + 30.127;
   1:  PR[91,3] = PR[90,3] + 105.095;
   1:L PR[91] R[100]mm/sec CNT100;
   1:  PR[91,1] = PR[90,1] + 33.248;
   1:  PR[91,2] = PR[90,2] + 30.548;
   1:  PR[91,3] = PR[90,3] + 105.101;
   1:L PR[91] R[100]mm/sec CNT100;
   1:  PR[91,1] = PR[90,1] + 31.709;
   1:  PR[91,2] = PR[90,2] + 30.581;
   1:  PR[91,3] = PR[90,3] + 105.121;
   1:L PR[91] R[100]mm/sec CNT100;
   1:  PR[91,1] = PR[90,1] + 27.915;
   1:  PR[91,2] = PR[90,2] + 30.327;
   1:  PR[91,3] = PR[90,3] + 105.128;
   1:L PR[91] R[100]mm/sec CNT100;
   1:  PR[91,1] = PR[90,1] + 26.644;
   1:  PR[91,2] = PR[90,2] + 30.180;
   1:  PR[91,3] = PR[90,3] + 105.147;
   1:L PR[91] R[100]mm/sec CNT100;
   1:  PR[91,1] = PR[90,1] + 26.104;
   1:  PR[91,2] = PR[90,2] + 30.092;
   1:  PR[91,3] = PR[90,3] + 105.153;
   1:L PR[91] R[100]mm/sec CNT100;
   1:  PR[91,1] = PR[90,1] + 25.544;
   1:  PR[91,2] = PR[90,2] + 30.107;
   1:  PR[91,3] = PR[90,3] + 105.155;
   1:L PR[91] R[100]mm/sec CNT100;
   1:  PR[91,1] = PR[90,1] + 24.329;
   1:  PR[91,2] = PR[90,2] + 30.087;
   1:  PR[91,3] = PR[90,3] + 105.158;
   1:L PR[91] R[100]mm/sec CNT100;
   1:  PR[91,1] = PR[90,1] + 15.055;
   1:  PR[91,2] = PR[90,2] + 29.482;
   1:  PR[91,3] = PR[90,3] + 105.164;
   1:L PR[91] R[100]mm/sec CNT100;
   1:  PR[91,1] = PR[90,1] + 14.674;
   1:  PR[91,2] = PR[90,2] + 29.410;
   1:  PR[91,3] = PR[90,3] + 105.209;
   1:L PR[91] R[100]mm/sec CNT100;
   1:  PR[91,1] = PR[90,1] + 6.614;
   1:  PR[91,2] = PR[90,2] + 28.195;
   1:  PR[91,3] = PR[90,3] + 105.211;
   1:L PR[91] R[100]mm/sec CNT100;
   1:  PR[91,1] = PR[90,1] + 2.021;
   1:  PR[91,2] = PR[90,2] + 27.161;
   1:  PR[91,3] = PR[90,3] + 105.251;
   1:L PR[91] R[100]mm/sec CNT100;
   1:  PR[91,1] = PR[90,1] + -0.771;
   1:  PR[91,2] = PR[90,2] + 26.651;
   1:  PR[91,3] = PR[90,3] + 105.273;
   1:L PR[91] R[100]mm/sec CNT100;
   1:  PR[91,1] = PR[90,1] + -9.843;
   1:  PR[91,2] = PR[90,2] + 24.252;
   1:  PR[91,3] = PR[90,3] + 105.287;
   1:L PR[91] R[100]mm/sec CNT100;
   1:  PR[91,1] = PR[90,1] + -17.871;
   1:  PR[91,2] = PR[90,2] + 21.371;
   1:  PR[91,3] = PR[90,3] + 105.333;
   1:L PR[91] R[100]mm/sec CNT100;
   1:  PR[91,1] = PR[90,1] + -24.750;
   1:  PR[91,2] = PR[90,2] + 18.099;
   1:  PR[91,3] = PR[90,3] + 105.374;
   1:L PR[91] R[100]mm/sec CNT100;
   1:  PR[91,1] = PR[90,1] + -30.389;
   1:  PR[91,2] = PR[90,2] + 14.529;
   1:  PR[91,3] = PR[90,3] + 105.411;
   1:L PR[91] R[100]mm/sec CNT100;
   1:  PR[91,1] = PR[90,1] + -34.749;
   1:  PR[91,2] = PR[90,2] + 10.761;
   1:  PR[91,3] = PR[90,3] + 105.443;
   1:L PR[91] R[100]mm/sec CNT100;
   1:  PR[91,1] = PR[90,1] + -37.797;
   1:  PR[91,2] = PR[90,2] + 6.911;
   1:  PR[91,3] = PR[90,3] + 105.471;
   1:L PR[91] R[100]mm/sec CNT100;
   1:  PR[91] = PR[90];
   1:  PR[91,1] = PR[90,1] + -37.438;
   1:  PR[91,2] = PR[90,2] + 3.095;
   1:  PR[91,3] = PR[90,3] + 106.795;
   1:L PR[91] R[100]mm/sec CNT100;
   1:  PR[91,1] = PR[90,1] + -38.021;
   1:  PR[91,2] = PR[90,2] + -0.729;
   1:  PR[91,3] = PR[90,3] + 105.516;
   1:L PR[91] R[100]mm/sec CNT100;
   1:  PR[91,1] = PR[90,1] + -37.438;
   1:  PR[91,2] = PR[90,2] + -4.554;
   1:  PR[91,3] = PR[90,3] + 105.535;
   1:L PR[91] R[100]mm/sec CNT100;
   1:  PR[91,1] = PR[90,1] + -35.649;
   1:  PR[91,2] = PR[90,2] + -8.432;
   1:  PR[91,3] = PR[90,3] + 105.554;
   1:L PR[91] R[100]mm/sec CNT100;
   1:  PR[91,1] = PR[90,1] + -32.577;
   1:  PR[91,2] = PR[90,2] + -12.315;
   1:  PR[91,3] = PR[90,3] + 105.575;
   1:L PR[91] R[100]mm/sec CNT100;
   1:  PR[91,1] = PR[90,1] + -31.486;
   1:  PR[91,2] = PR[90,2] + -13.265;
   1:  PR[91,3] = PR[90,3] + 105.599;
   1:L PR[91] R[100]mm/sec CNT100;
   1:  PR[91,1] = PR[90,1] + -28.191;
   1:  PR[91,2] = PR[90,2] + -16.108;
   1:  PR[91,3] = PR[90,3] + 105.606;
   1:L PR[91] R[100]mm/sec CNT100;
   1:  PR[91,1] = PR[90,1] + -22.512;
   1:  PR[91,2] = PR[90,2] + -19.706;
   1:  PR[91,3] = PR[90,3] + 105.628;
   1:L PR[91] R[100]mm/sec CNT100;
   1:  PR[91,1] = PR[90,1] + -15.586;
   1:  PR[91,2] = PR[90,2] + -23.002;
   1:  PR[91,3] = PR[90,3] + 105.660;
   1:L PR[91] R[100]mm/sec CNT100;
   1:  PR[91,1] = PR[90,1] + -7.503;
   1:  PR[91,2] = PR[90,2] + -25.906;
   1:  PR[91,3] = PR[90,3] + 105.698;
   1:L PR[91] R[100]mm/sec CNT100;
   1:  PR[91,1] = PR[90,1] + 1.762;
   1:  PR[91,2] = PR[90,2] + -28.366;
   1:  PR[91,3] = PR[90,3] + 105.740;
   1:L PR[91] R[100]mm/sec CNT100;
   1:  PR[91,1] = PR[90,1] + 7.941;
   1:  PR[91,2] = PR[90,2] + -29.756;
   1:  PR[91,3] = PR[90,3] + 105.787;
   1:L PR[91] R[100]mm/sec CNT100;
   1:  PR[91,1] = PR[90,1] + 13.802;
   1:  PR[91,2] = PR[90,2] + -30.639;
   1:  PR[91,3] = PR[90,3] + 105.818;
   1:L PR[91] R[100]mm/sec CNT100;
   1:  PR[91,1] = PR[90,1] + 16.569;
   1:  PR[91,2] = PR[90,2] + -31.163;
   1:  PR[91,3] = PR[90,3] + 105.847;
   1:L PR[91] R[100]mm/sec CNT100;
   1:  PR[91,1] = PR[90,1] + 25.855;
   1:  PR[91,2] = PR[90,2] + -31.775;
   1:  PR[91,3] = PR[90,3] + 105.861;
   1:L PR[91] R[100]mm/sec CNT100;
   1:  PR[91,1] = PR[90,1] + 26.725;
   1:  PR[91,2] = PR[90,2] + -31.791;
   1:  PR[91,3] = PR[90,3] + 105.907;
   1:L PR[91] R[100]mm/sec CNT100;
   1:  PR[91,1] = PR[90,1] + 27.669;
   1:  PR[91,2] = PR[90,2] + -31.899;
   1:  PR[91,3] = PR[90,3] + 105.911;
   1:L PR[91] R[100]mm/sec CNT100;
   1:  PR[91,1] = PR[90,1] + 32.407;
   1:  PR[91,2] = PR[90,2] + -32.212;
   1:  PR[91,3] = PR[90,3] + 105.916;
   1:L PR[91] R[100]mm/sec CNT100;
   1:  PR[91,1] = PR[90,1] + 32.895;
   1:  PR[91,2] = PR[90,2] + -32.202;
   1:  PR[91,3] = PR[90,3] + 105.939;
   1:L PR[91] R[100]mm/sec CNT100;
   1:  PR[91,1] = PR[90,1] + 38.092;
   1:  PR[91,2] = PR[90,2] + -31.668;
   1:  PR[91,3] = PR[90,3] + 105.941;
   1:L PR[91] R[100]mm/sec CNT100;
   1:  PR[91,1] = PR[90,1] + 43.282;
   1:  PR[91,2] = PR[90,2] + -30.250;
   1:  PR[91,3] = PR[90,3] + 105.967;
   1:L PR[91] R[100]mm/sec CNT100;
   1:  PR[91,1] = PR[90,1] + 43.736;
   1:  PR[91,2] = PR[90,2] + -30.088;
   1:  PR[91,3] = PR[90,3] + 105.993;
   1:L PR[91] R[100]mm/sec CNT100;
   1:  PR[91,1] = PR[90,1] + 48.043;
   1:  PR[91,2] = PR[90,2] + -28.096;
   1:  PR[91,3] = PR[90,3] + 105.996;
   1:L PR[91] R[100]mm/sec CNT100;
   1:  PR[91,1] = PR[90,1] + 49.407;
   1:  PR[91,2] = PR[90,2] + -27.311;
   1:  PR[91,3] = PR[90,3] + 106.019;
   1:L PR[91] R[100]mm/sec CNT100;
   1:  PR[91,1] = PR[90,1] + 52.446;
   1:  PR[91,2] = PR[90,2] + -25.229;
   1:  PR[91,3] = PR[90,3] + 106.027;
   1:L PR[91] R[100]mm/sec CNT100;
   1:  PR[91,1] = PR[90,1] + 54.789;
   1:  PR[91,2] = PR[90,2] + -23.251;
   1:  PR[91,3] = PR[90,3] + 106.045;
   1:L PR[91] R[100]mm/sec CNT100;
   1:  PR[91,1] = PR[90,1] + 56.409;
   1:  PR[91,2] = PR[90,2] + -21.678;
   1:  PR[91,3] = PR[90,3] + 106.060;
   1:L PR[91] R[100]mm/sec CNT100;
   1:  PR[91,1] = PR[90,1] + 59.575;
   1:  PR[91,2] = PR[90,2] + -17.816;
   1:  PR[91,3] = PR[90,3] + 106.071;
   1:L PR[91] R[100]mm/sec CNT100;
   1:  PR[91,1] = PR[90,1] + 59.849;
   1:  PR[91,2] = PR[90,2] + -17.438;
   1:  PR[91,3] = PR[90,3] + 106.095;
   1:L PR[91] R[100]mm/sec CNT100;
   1:  PR[91,1] = PR[90,1] + 60.871;
   1:  PR[91,2] = PR[90,2] + -15.568;
   1:  PR[91,3] = PR[90,3] + 106.098;
   1:L PR[91] R[100]mm/sec CNT100;
   1:  PR[91,1] = PR[90,1] + 62.396;
   1:  PR[91,2] = PR[90,2] + -12.864;
   1:  PR[91,3] = PR[90,3] + 106.108;
   1:L PR[91] R[100]mm/sec CNT100;
   1:  PR[91,1] = PR[90,1] + 62.780;
   1:  PR[91,2] = PR[90,2] + -12.209;
   1:  PR[91,3] = PR[90,3] + 106.123;
   1:L PR[91] R[100]mm/sec CNT100;
   1:  PR[91,1] = PR[90,1] + 63.948;
   1:  PR[91,2] = PR[90,2] + -8.607;
   1:  PR[91,3] = PR[90,3] + 106.127;
   1:L PR[91] R[100]mm/sec CNT100;
   1:  PR[91,1] = PR[90,1] + 64.641;
   1:  PR[91,2] = PR[90,2] + -6.555;
   1:  PR[91,3] = PR[90,3] + 106.146;
   1:L PR[91] R[100]mm/sec CNT100;
   1:  PR[91,1] = PR[90,1] + 65.278;
   1:  PR[91,2] = PR[90,2] + -0.729;
   1:  PR[91,3] = PR[90,3] + 106.156;
   1:L PR[91] R[100]mm/sec CNT100;
   1:  PR[91,1] = PR[90,1] + 64.641;
   1:  PR[91,2] = PR[90,2] + 5.096;
   1:  PR[91,3] = PR[90,3] + 106.185;
   1:L PR[91] R[100]mm/sec CNT100;
   1:  PR[91,1] = PR[90,1] + 63.948;
   1:  PR[91,2] = PR[90,2] + 7.149;
   1:  PR[91,3] = PR[90,3] + 106.214;
   1:L PR[91] R[100]mm/sec CNT100;
   1:  PR[91,1] = PR[90,1] + 62.780;
   1:  PR[91,2] = PR[90,2] + 10.749;
   1:  PR[91,3] = PR[90,3] + 106.224;
   1:L PR[91] R[100]mm/sec CNT100;
   1:  PR[91,1] = PR[90,1] + 62.396;
   1:  PR[91,2] = PR[90,2] + 11.404;
   1:  PR[91,3] = PR[90,3] + 106.243;
   1:L PR[91] R[100]mm/sec CNT100;
   1:  PR[91,1] = PR[90,1] + 60.871;
   1:  PR[91,2] = PR[90,2] + 14.110;
   1:  PR[91,3] = PR[90,3] + 106.247;
   1:L PR[91] R[100]mm/sec CNT100;
   1:  PR[91,1] = PR[90,1] + 59.850;
   1:  PR[91,2] = PR[90,2] + 15.978;
   1:  PR[91,3] = PR[90,3] + 106.262;
   1:L PR[91] R[100]mm/sec CNT100;
   1:  PR[91,1] = PR[90,1] + 59.576;
   1:  PR[91,2] = PR[90,2] + 16.356;
   1:  PR[91,3] = PR[90,3] + 106.272;
   1:L PR[91] R[100]mm/sec CNT100;
   1:  PR[91,1] = PR[90,1] + 56.408;
   1:  PR[91,2] = PR[90,2] + 20.220;
   1:  PR[91,3] = PR[90,3] + 106.274;
   1:L PR[91] R[100]mm/sec CNT100;
   1:  PR[91,1] = PR[90,1] + 54.786;
   1:  PR[91,2] = PR[90,2] + 21.794;
   1:  PR[91,3] = PR[90,3] + 106.299;
   1:L PR[91] R[100]mm/sec CNT100;
   1:  PR[91,1] = PR[90,1] + 52.441;
   1:  PR[91,2] = PR[90,2] + 23.774;
   1:  PR[91,3] = PR[90,3] + 106.310;
   1:L PR[91] R[100]mm/sec CNT100;
   1:  PR[91,1] = PR[90,1] + 49.399;
   1:  PR[91,2] = PR[90,2] + 25.857;
   1:  PR[91,3] = PR[90,3] + 106.325;
   1:L PR[91] R[100]mm/sec CNT100;
   1:  PR[91,1] = PR[90,1] + 48.034;
   1:  PR[91,2] = PR[90,2] + 26.643;
   1:  PR[91,3] = PR[90,3] + 106.343;
   1:L PR[91] R[100]mm/sec CNT100;
   1:  PR[91,1] = PR[90,1] + 43.721;
   1:  PR[91,2] = PR[90,2] + 28.634;
   1:  PR[91,3] = PR[90,3] + 106.351;
   1:L PR[91] R[100]mm/sec CNT100;
   1:  PR[91,1] = PR[90,1] + 43.269;
   1:  PR[91,2] = PR[90,2] + 28.796;
   1:  PR[91,3] = PR[90,3] + 106.374;
   1:L PR[91] R[100]mm/sec CNT100;
   1:  PR[91,1] = PR[90,1] + 38.028;
   1:  PR[91,2] = PR[90,2] + 30.218;
   1:  PR[91,3] = PR[90,3] + 106.377;
   1:L PR[91] R[100]mm/sec CNT100;
   1:  PR[91,1] = PR[90,1] + 32.877;
   1:  PR[91,2] = PR[90,2] + 30.743;
   1:  PR[91,3] = PR[90,3] + 106.403;
   1:L PR[91] R[100]mm/sec CNT100;
   1:  PR[91,1] = PR[90,1] + 32.386;
   1:  PR[91,2] = PR[90,2] + 30.754;
   1:  PR[91,3] = PR[90,3] + 106.429;
   1:L PR[91] R[100]mm/sec CNT100;
   1:  PR[91,1] = PR[90,1] + 27.651;
   1:  PR[91,2] = PR[90,2] + 30.438;
   1:  PR[91,3] = PR[90,3] + 106.431;
   1:L PR[91] R[100]mm/sec CNT100;
   1:  PR[91,1] = PR[90,1] + 26.723;
   1:  PR[91,2] = PR[90,2] + 30.330;
   1:  PR[91,3] = PR[90,3] + 106.454;
   1:L PR[91] R[100]mm/sec CNT100;
   1:  PR[91,1] = PR[90,1] + 25.868;
   1:  PR[91,2] = PR[90,2] + 30.317;
   1:  PR[91,3] = PR[90,3] + 106.459;
   1:L PR[91] R[100]mm/sec CNT100;
   1:  PR[91,1] = PR[90,1] + 16.575;
   1:  PR[91,2] = PR[90,2] + 29.705;
   1:  PR[91,3] = PR[90,3] + 106.463;
   1:L PR[91] R[100]mm/sec CNT100;
   1:  PR[91,1] = PR[90,1] + 13.802;
   1:  PR[91,2] = PR[90,2] + 29.181;
   1:  PR[91,3] = PR[90,3] + 106.509;
   1:L PR[91] R[100]mm/sec CNT100;
   1:  PR[91,1] = PR[90,1] + 7.941;
   1:  PR[91,2] = PR[90,2] + 28.297;
   1:  PR[91,3] = PR[90,3] + 106.523;
   1:L PR[91] R[100]mm/sec CNT100;
   1:  PR[91,1] = PR[90,1] + 1.762;
   1:  PR[91,2] = PR[90,2] + 26.907;
   1:  PR[91,3] = PR[90,3] + 106.552;
   1:L PR[91] R[100]mm/sec CNT100;
   1:  PR[91,1] = PR[90,1] + -7.503;
   1:  PR[91,2] = PR[90,2] + 24.448;
   1:  PR[91,3] = PR[90,3] + 106.583;
   1:L PR[91] R[100]mm/sec CNT100;
   1:  PR[91,1] = PR[90,1] + -15.586;
   1:  PR[91,2] = PR[90,2] + 21.544;
   1:  PR[91,3] = PR[90,3] + 106.630;
   1:L PR[91] R[100]mm/sec CNT100;
   1:  PR[91,1] = PR[90,1] + -22.512;
   1:  PR[91,2] = PR[90,2] + 18.247;
   1:  PR[91,3] = PR[90,3] + 106.672;
   1:L PR[91] R[100]mm/sec CNT100;
   1:  PR[91,1] = PR[90,1] + -28.190;
   1:  PR[91,2] = PR[90,2] + 14.650;
   1:  PR[91,3] = PR[90,3] + 106.709;
   1:L PR[91] R[100]mm/sec CNT100;
   1:  PR[91,1] = PR[90,1] + -32.579;
   1:  PR[91,2] = PR[90,2] + 10.853;
   1:  PR[91,3] = PR[90,3] + 106.742;
   1:L PR[91] R[100]mm/sec CNT100;
   1:  PR[91,1] = PR[90,1] + -35.649;
   1:  PR[91,2] = PR[90,2] + 6.973;
   1:  PR[91,3] = PR[90,3] + 106.771;
   1:L PR[91] R[100]mm/sec CNT100;
   1:  PR[91] = PR[90];
   1:  PR[91,1] = PR[90,1] + -35.303;
   1:  PR[91,2] = PR[90,2] + 3.126;
   1:  PR[91,3] = PR[90,3] + 108.095;
   1:L PR[91] R[100]mm/sec CNT100;
   1:  PR[91,1] = PR[90,1] + -35.891;
   1:  PR[91,2] = PR[90,2] + -0.729;
   1:  PR[91,3] = PR[90,3] + 106.816;
   1:L PR[91] R[100]mm/sec CNT100;
   1:  PR[91,1] = PR[90,1] + -35.303;
   1:  PR[91,2] = PR[90,2] + -4.585;
   1:  PR[91,3] = PR[90,3] + 106.836;
   1:L PR[91] R[100]mm/sec CNT100;
   1:  PR[91,1] = PR[90,1] + -33.501;
   1:  PR[91,2] = PR[90,2] + -8.494;
   1:  PR[91,3] = PR[90,3] + 106.855;
   1:L PR[91] R[100]mm/sec CNT100;
   1:  PR[91,1] = PR[90,1] + -30.408;
   1:  PR[91,2] = PR[90,2] + -12.406;
   1:  PR[91,3] = PR[90,3] + 106.876;
   1:L PR[91] R[100]mm/sec CNT100;
   1:  PR[91,1] = PR[90,1] + -28.966;
   1:  PR[91,2] = PR[90,2] + -13.661;
   1:  PR[91,3] = PR[90,3] + 106.901;
   1:L PR[91] R[100]mm/sec CNT100;
   1:  PR[91,1] = PR[90,1] + -25.991;
   1:  PR[91,2] = PR[90,2] + -16.228;
   1:  PR[91,3] = PR[90,3] + 106.910;
   1:L PR[91] R[100]mm/sec CNT100;
   1:  PR[91,1] = PR[90,1] + -20.274;
   1:  PR[91,2] = PR[90,2] + -19.853;
   1:  PR[91,3] = PR[90,3] + 106.930;
   1:L PR[91] R[100]mm/sec CNT100;
   1:  PR[91,1] = PR[90,1] + -13.301;
   1:  PR[91,2] = PR[90,2] + -23.175;
   1:  PR[91,3] = PR[90,3] + 106.963;
   1:L PR[91] R[100]mm/sec CNT100;
   1:  PR[91,1] = PR[90,1] + -5.165;
   1:  PR[91,2] = PR[90,2] + -26.102;
   1:  PR[91,3] = PR[90,3] + 107.001;
   1:L PR[91] R[100]mm/sec CNT100;
   1:  PR[91,1] = PR[90,1] + 0.887;
   1:  PR[91,2] = PR[90,2] + -27.704;
   1:  PR[91,3] = PR[90,3] + 107.044;
   1:L PR[91] R[100]mm/sec CNT100;
   1:  PR[91,1] = PR[90,1] + 2.723;
   1:  PR[91,2] = PR[90,2] + -28.294;
   1:  PR[91,3] = PR[90,3] + 107.075;
   1:L PR[91] R[100]mm/sec CNT100;
   1:  PR[91,1] = PR[90,1] + 5.426;
   1:  PR[91,2] = PR[90,2] + -28.994;
   1:  PR[91,3] = PR[90,3] + 107.085;
   1:L PR[91] R[100]mm/sec CNT100;
   1:  PR[91,1] = PR[90,1] + 9.267;
   1:  PR[91,2] = PR[90,2] + -29.858;
   1:  PR[91,3] = PR[90,3] + 107.098;
   1:L PR[91] R[100]mm/sec CNT100;
   1:  PR[91,1] = PR[90,1] + 12.931;
   1:  PR[91,2] = PR[90,2] + -30.410;
   1:  PR[91,3] = PR[90,3] + 107.118;
   1:L PR[91] R[100]mm/sec CNT100;
   1:  PR[91,1] = PR[90,1] + 18.085;
   1:  PR[91,2] = PR[90,2] + -31.386;
   1:  PR[91,3] = PR[90,3] + 107.136;
   1:L PR[91] R[100]mm/sec CNT100;
   1:  PR[91,1] = PR[90,1] + 32.755;
   1:  PR[91,2] = PR[90,2] + -32.361;
   1:  PR[91,3] = PR[90,3] + 107.162;
   1:L PR[91] R[100]mm/sec CNT100;
   1:  PR[91,1] = PR[90,1] + 33.002;
   1:  PR[91,2] = PR[90,2] + -32.363;
   1:  PR[91,3] = PR[90,3] + 107.235;
   1:L PR[91] R[100]mm/sec CNT100;
   1:  PR[91,1] = PR[90,1] + 37.963;
   1:  PR[91,2] = PR[90,2] + -31.870;
   1:  PR[91,3] = PR[90,3] + 107.236;
   1:L PR[91] R[100]mm/sec CNT100;
   1:  PR[91,1] = PR[90,1] + 38.977;
   1:  PR[91,2] = PR[90,2] + -31.699;
   1:  PR[91,3] = PR[90,3] + 107.261;
   1:L PR[91] R[100]mm/sec CNT100;
   1:  PR[91,1] = PR[90,1] + 43.040;
   1:  PR[91,2] = PR[90,2] + -30.595;
   1:  PR[91,3] = PR[90,3] + 107.266;
   1:L PR[91] R[100]mm/sec CNT100;
   1:  PR[91,1] = PR[90,1] + 45.009;
   1:  PR[91,2] = PR[90,2] + -29.889;
   1:  PR[91,3] = PR[90,3] + 107.287;
   1:L PR[91] R[100]mm/sec CNT100;
   1:  PR[91,1] = PR[90,1] + 47.878;
   1:  PR[91,2] = PR[90,2] + -28.562;
   1:  PR[91,3] = PR[90,3] + 107.297;
   1:L PR[91] R[100]mm/sec CNT100;
   1:  PR[91,1] = PR[90,1] + 50.965;
   1:  PR[91,2] = PR[90,2] + -26.786;
   1:  PR[91,3] = PR[90,3] + 107.313;
   1:L PR[91] R[100]mm/sec CNT100;
   1:  PR[91,1] = PR[90,1] + 52.399;
   1:  PR[91,2] = PR[90,2] + -25.803;
   1:  PR[91,3] = PR[90,3] + 107.330;
   1:L PR[91] R[100]mm/sec CNT100;
   1:  PR[91,1] = PR[90,1] + 56.564;
   1:  PR[91,2] = PR[90,2] + -22.286;
   1:  PR[91,3] = PR[90,3] + 107.339;
   1:L PR[91] R[100]mm/sec CNT100;
   1:  PR[91,1] = PR[90,1] + 59.657;
   1:  PR[91,2] = PR[90,2] + -18.639;
   1:  PR[91,3] = PR[90,3] + 107.366;
   1:L PR[91] R[100]mm/sec CNT100;
   1:  PR[91,1] = PR[90,1] + 60.635;
   1:  PR[91,2] = PR[90,2] + -17.521;
   1:  PR[91,3] = PR[90,3] + 107.389;
   1:L PR[91] R[100]mm/sec CNT100;
   1:  PR[91,1] = PR[90,1] + 61.969;
   1:  PR[91,2] = PR[90,2] + -15.155;
   1:  PR[91,3] = PR[90,3] + 107.397;
   1:L PR[91] R[100]mm/sec CNT100;
   1:  PR[91,1] = PR[90,1] + 63.685;
   1:  PR[91,2] = PR[90,2] + -12.224;
   1:  PR[91,3] = PR[90,3] + 107.410;
   1:L PR[91] R[100]mm/sec CNT100;
   1:  PR[91,1] = PR[90,1] + 64.460;
   1:  PR[91,2] = PR[90,2] + -9.904;
   1:  PR[91,3] = PR[90,3] + 107.427;
   1:L PR[91] R[100]mm/sec CNT100;
   1:  PR[91,1] = PR[90,1] + 65.455;
   1:  PR[91,2] = PR[90,2] + -7.038;
   1:  PR[91,3] = PR[90,3] + 107.439;
   1:L PR[91] R[100]mm/sec CNT100;
   1:  PR[91,1] = PR[90,1] + 65.654;
   1:  PR[91,2] = PR[90,2] + -6.234;
   1:  PR[91,3] = PR[90,3] + 107.454;
   1:L PR[91] R[100]mm/sec CNT100;
   1:  PR[91,1] = PR[90,1] + 66.079;
   1:  PR[91,2] = PR[90,2] + -2.515;
   1:  PR[91,3] = PR[90,3] + 107.458;
   1:L PR[91] R[100]mm/sec CNT100;
   1:  PR[91,1] = PR[90,1] + 66.226;
   1:  PR[91,2] = PR[90,2] + -0.755;
   1:  PR[91,3] = PR[90,3] + 107.477;
   1:L PR[91] R[100]mm/sec CNT100;
   1:  PR[91,1] = PR[90,1] + 65.763;
   1:  PR[91,2] = PR[90,2] + 3.477;
   1:  PR[91,3] = PR[90,3] + 107.485;
   1:L PR[91] R[100]mm/sec CNT100;
   1:  PR[91,1] = PR[90,1] + 65.647;
   1:  PR[91,2] = PR[90,2] + 4.802;
   1:  PR[91,3] = PR[90,3] + 107.507;
   1:L PR[91] R[100]mm/sec CNT100;
   1:  PR[91,1] = PR[90,1] + 65.455;
   1:  PR[91,2] = PR[90,2] + 5.580;
   1:  PR[91,3] = PR[90,3] + 107.513;
   1:L PR[91] R[100]mm/sec CNT100;
   1:  PR[91,1] = PR[90,1] + 64.460;
   1:  PR[91,2] = PR[90,2] + 8.445;
   1:  PR[91,3] = PR[90,3] + 107.517;
   1:L PR[91] R[100]mm/sec CNT100;
   1:  PR[91,1] = PR[90,1] + 63.684;
   1:  PR[91,2] = PR[90,2] + 10.767;
   1:  PR[91,3] = PR[90,3] + 107.532;
   1:L PR[91] R[100]mm/sec CNT100;
   1:  PR[91,1] = PR[90,1] + 61.969;
   1:  PR[91,2] = PR[90,2] + 13.697;
   1:  PR[91,3] = PR[90,3] + 107.544;
   1:L PR[91] R[100]mm/sec CNT100;
   1:  PR[91,1] = PR[90,1] + 60.635;
   1:  PR[91,2] = PR[90,2] + 16.062;
   1:  PR[91,3] = PR[90,3] + 107.561;
   1:L PR[91] R[100]mm/sec CNT100;
   1:  PR[91,1] = PR[90,1] + 59.657;
   1:  PR[91,2] = PR[90,2] + 17.180;
   1:  PR[91,3] = PR[90,3] + 107.574;
   1:L PR[91] R[100]mm/sec CNT100;
   1:  PR[91,1] = PR[90,1] + 56.587;
   1:  PR[91,2] = PR[90,2] + 20.805;
   1:  PR[91,3] = PR[90,3] + 107.582;
   1:L PR[91] R[100]mm/sec CNT100;
   1:  PR[91,1] = PR[90,1] + 52.398;
   1:  PR[91,2] = PR[90,2] + 24.345;
   1:  PR[91,3] = PR[90,3] + 107.605;
   1:L PR[91] R[100]mm/sec CNT100;
   1:  PR[91,1] = PR[90,1] + 50.963;
   1:  PR[91,2] = PR[90,2] + 25.328;
   1:  PR[91,3] = PR[90,3] + 107.632;
   1:L PR[91] R[100]mm/sec CNT100;
   1:  PR[91,1] = PR[90,1] + 47.874;
   1:  PR[91,2] = PR[90,2] + 27.106;
   1:  PR[91,3] = PR[90,3] + 107.641;
   1:L PR[91] R[100]mm/sec CNT100;
   1:  PR[91,1] = PR[90,1] + 45.001;
   1:  PR[91,2] = PR[90,2] + 28.433;
   1:  PR[91,3] = PR[90,3] + 107.659;
   1:L PR[91] R[100]mm/sec CNT100;
   1:  PR[91,1] = PR[90,1] + 43.031;
   1:  PR[91,2] = PR[90,2] + 29.139;
   1:  PR[91,3] = PR[90,3] + 107.674;
   1:L PR[91] R[100]mm/sec CNT100;
   1:  PR[91,1] = PR[90,1] + 38.962;
   1:  PR[91,2] = PR[90,2] + 30.243;
   1:  PR[91,3] = PR[90,3] + 107.685;
   1:L PR[91] R[100]mm/sec CNT100;
   1:  PR[91,1] = PR[90,1] + 37.948;
   1:  PR[91,2] = PR[90,2] + 30.414;
   1:  PR[91,3] = PR[90,3] + 107.705;
   1:L PR[91] R[100]mm/sec CNT100;
   1:  PR[91,1] = PR[90,1] + 32.980;
   1:  PR[91,2] = PR[90,2] + 30.905;
   1:  PR[91,3] = PR[90,3] + 107.710;
   1:L PR[91] R[100]mm/sec CNT100;
   1:  PR[91,1] = PR[90,1] + 32.734;
   1:  PR[91,2] = PR[90,2] + 30.903;
   1:  PR[91,3] = PR[90,3] + 107.735;
   1:L PR[91] R[100]mm/sec CNT100;
   1:  PR[91,1] = PR[90,1] + 18.096;
   1:  PR[91,2] = PR[90,2] + 29.928;
   1:  PR[91,3] = PR[90,3] + 107.736;
   1:L PR[91] R[100]mm/sec CNT100;
   1:  PR[91,1] = PR[90,1] + 12.931;
   1:  PR[91,2] = PR[90,2] + 28.952;
   1:  PR[91,3] = PR[90,3] + 107.809;
   1:L PR[91] R[100]mm/sec CNT100;
   1:  PR[91,1] = PR[90,1] + 9.268;
   1:  PR[91,2] = PR[90,2] + 28.399;
   1:  PR[91,3] = PR[90,3] + 107.835;
   1:L PR[91] R[100]mm/sec CNT100;
   1:  PR[91,1] = PR[90,1] + 5.427;
   1:  PR[91,2] = PR[90,2] + 27.535;
   1:  PR[91,3] = PR[90,3] + 107.853;
   1:L PR[91] R[100]mm/sec CNT100;
   1:  PR[91,1] = PR[90,1] + 2.723;
   1:  PR[91,2] = PR[90,2] + 26.836;
   1:  PR[91,3] = PR[90,3] + 107.873;
   1:L PR[91] R[100]mm/sec CNT100;
   1:  PR[91,1] = PR[90,1] + 0.887;
   1:  PR[91,2] = PR[90,2] + 26.246;
   1:  PR[91,3] = PR[90,3] + 107.887;
   1:L PR[91] R[100]mm/sec CNT100;
   1:  PR[91,1] = PR[90,1] + -5.165;
   1:  PR[91,2] = PR[90,2] + 24.643;
   1:  PR[91,3] = PR[90,3] + 107.896;
   1:L PR[91] R[100]mm/sec CNT100;
   1:  PR[91,1] = PR[90,1] + -13.301;
   1:  PR[91,2] = PR[90,2] + 21.717;
   1:  PR[91,3] = PR[90,3] + 107.927;
   1:L PR[91] R[100]mm/sec CNT100;
   1:  PR[91,1] = PR[90,1] + -20.276;
   1:  PR[91,2] = PR[90,2] + 18.394;
   1:  PR[91,3] = PR[90,3] + 107.970;
   1:L PR[91] R[100]mm/sec CNT100;
   1:  PR[91,1] = PR[90,1] + -23.310;
   1:  PR[91,2] = PR[90,2] + 16.479;
   1:  PR[91,3] = PR[90,3] + 108.008;
   1:L PR[91] R[100]mm/sec CNT100;
   1:  PR[91,1] = PR[90,1] + -25.988;
   1:  PR[91,2] = PR[90,2] + 14.772;
   1:  PR[91,3] = PR[90,3] + 108.026;
   1:L PR[91] R[100]mm/sec CNT100;
   1:  PR[91,1] = PR[90,1] + -30.410;
   1:  PR[91,2] = PR[90,2] + 10.945;
   1:  PR[91,3] = PR[90,3] + 108.041;
   1:L PR[91] R[100]mm/sec CNT100;
   1:  PR[91,1] = PR[90,1] + -33.501;
   1:  PR[91,2] = PR[90,2] + 7.035;
   1:  PR[91,3] = PR[90,3] + 108.070;
   1:L PR[91] R[100]mm/sec CNT100;
   1:  PR[91] = PR[90];
   1:  PR[91,1] = PR[90,1] + -33.168;
   1:  PR[91,2] = PR[90,2] + 3.157;
   1:  PR[91,3] = PR[90,3] + 109.395;
   1:L PR[91] R[100]mm/sec CNT100;
   1:  PR[91,1] = PR[90,1] + -33.760;
   1:  PR[91,2] = PR[90,2] + -0.729;
   1:  PR[91,3] = PR[90,3] + 108.117;
   1:L PR[91] R[100]mm/sec CNT100;
   1:  PR[91,1] = PR[90,1] + -33.168;
   1:  PR[91,2] = PR[90,2] + -4.616;
   1:  PR[91,3] = PR[90,3] + 108.136;
   1:L PR[91] R[100]mm/sec CNT100;
   1:  PR[91,1] = PR[90,1] + -31.353;
   1:  PR[91,2] = PR[90,2] + -8.556;
   1:  PR[91,3] = PR[90,3] + 108.156;
   1:L PR[91] R[100]mm/sec CNT100;
   1:  PR[91,1] = PR[90,1] + -28.238;
   1:  PR[91,2] = PR[90,2] + -12.497;
   1:  PR[91,3] = PR[90,3] + 108.177;
   1:L PR[91] R[100]mm/sec CNT100;
   1:  PR[91,1] = PR[90,1] + -26.447;
   1:  PR[91,2] = PR[90,2] + -14.057;
   1:  PR[91,3] = PR[90,3] + 108.203;
   1:L PR[91] R[100]mm/sec CNT100;
   1:  PR[91,1] = PR[90,1] + -23.792;
   1:  PR[91,2] = PR[90,2] + -16.348;
   1:  PR[91,3] = PR[90,3] + 108.214;
   1:L PR[91] R[100]mm/sec CNT100;
   1:  PR[91,1] = PR[90,1] + -18.036;
   1:  PR[91,2] = PR[90,2] + -20.001;
   1:  PR[91,3] = PR[90,3] + 108.232;
   1:L PR[91] R[100]mm/sec CNT100;
   1:  PR[91,1] = PR[90,1] + -11.016;
   1:  PR[91,2] = PR[90,2] + -23.349;
   1:  PR[91,3] = PR[90,3] + 108.266;
   1:L PR[91] R[100]mm/sec CNT100;
   1:  PR[91,1] = PR[90,1] + -2.826;
   1:  PR[91,2] = PR[90,2] + -26.298;
   1:  PR[91,3] = PR[90,3] + 108.305;
   1:L PR[91] R[100]mm/sec CNT100;
   1:  PR[91,1] = PR[90,1] + 0.239;
   1:  PR[91,2] = PR[90,2] + -27.109;
   1:  PR[91,3] = PR[90,3] + 108.348;
   1:L PR[91] R[100]mm/sec CNT100;
   1:  PR[91,1] = PR[90,1] + 3.791;
   1:  PR[91,2] = PR[90,2] + -28.251;
   1:  PR[91,3] = PR[90,3] + 108.364;
   1:L PR[91] R[100]mm/sec CNT100;
   1:  PR[91,1] = PR[90,1] + 9.096;
   1:  PR[91,2] = PR[90,2] + -29.623;
   1:  PR[91,3] = PR[90,3] + 108.383;
   1:L PR[91] R[100]mm/sec CNT100;
   1:  PR[91,1] = PR[90,1] + 10.594;
   1:  PR[91,2] = PR[90,2] + -29.960;
   1:  PR[91,3] = PR[90,3] + 108.410;
   1:L PR[91] R[100]mm/sec CNT100;
   1:  PR[91,1] = PR[90,1] + 12.059;
   1:  PR[91,2] = PR[90,2] + -30.181;
   1:  PR[91,3] = PR[90,3] + 108.417;
   1:L PR[91] R[100]mm/sec CNT100;
   1:  PR[91,1] = PR[90,1] + 19.601;
   1:  PR[91,2] = PR[90,2] + -31.608;
   1:  PR[91,3] = PR[90,3] + 108.425;
   1:L PR[91] R[100]mm/sec CNT100;
   1:  PR[91,1] = PR[90,1] + 32.469;
   1:  PR[91,2] = PR[90,2] + -32.466;
   1:  PR[91,3] = PR[90,3] + 108.463;
   1:L PR[91] R[100]mm/sec CNT100;
   1:  PR[91,1] = PR[90,1] + 33.818;
   1:  PR[91,2] = PR[90,2] + -32.475;
   1:  PR[91,3] = PR[90,3] + 108.527;
   1:L PR[91] R[100]mm/sec CNT100;
   1:  PR[91,1] = PR[90,1] + 37.673;
   1:  PR[91,2] = PR[90,2] + -32.092;
   1:  PR[91,3] = PR[90,3] + 108.534;
   1:L PR[91] R[100]mm/sec CNT100;
   1:  PR[91,1] = PR[90,1] + 40.001;
   1:  PR[91,2] = PR[90,2] + -31.699;
   1:  PR[91,3] = PR[90,3] + 108.554;
   1:L PR[91] R[100]mm/sec CNT100;
   1:  PR[91,1] = PR[90,1] + 42.797;
   1:  PR[91,2] = PR[90,2] + -30.939;
   1:  PR[91,3] = PR[90,3] + 108.565;
   1:L PR[91] R[100]mm/sec CNT100;
   1:  PR[91,1] = PR[90,1] + 46.282;
   1:  PR[91,2] = PR[90,2] + -29.690;
   1:  PR[91,3] = PR[90,3] + 108.580;
   1:L PR[91] R[100]mm/sec CNT100;
   1:  PR[91,1] = PR[90,1] + 47.714;
   1:  PR[91,2] = PR[90,2] + -29.028;
   1:  PR[91,3] = PR[90,3] + 108.598;
   1:L PR[91] R[100]mm/sec CNT100;
   1:  PR[91,1] = PR[90,1] + 52.439;
   1:  PR[91,2] = PR[90,2] + -26.310;
   1:  PR[91,3] = PR[90,3] + 108.606;
   1:L PR[91] R[100]mm/sec CNT100;
   1:  PR[91,1] = PR[90,1] + 56.151;
   1:  PR[91,2] = PR[90,2] + -23.284;
   1:  PR[91,3] = PR[90,3] + 108.633;
   1:L PR[91] R[100]mm/sec CNT100;
   1:  PR[91,1] = PR[90,1] + 57.391;
   1:  PR[91,2] = PR[90,2] + -22.295;
   1:  PR[91,3] = PR[90,3] + 108.657;
   1:L PR[91] R[100]mm/sec CNT100;
   1:  PR[91,1] = PR[90,1] + 59.089;
   1:  PR[91,2] = PR[90,2] + -20.291;
   1:  PR[91,3] = PR[90,3] + 108.665;
   1:L PR[91] R[100]mm/sec CNT100;
   1:  PR[91,1] = PR[90,1] + 61.490;
   1:  PR[91,2] = PR[90,2] + -17.544;
   1:  PR[91,3] = PR[90,3] + 108.678;
   1:L PR[91] R[100]mm/sec CNT100;
   1:  PR[91,1] = PR[90,1] + 63.751;
   1:  PR[91,2] = PR[90,2] + -13.654;
   1:  PR[91,3] = PR[90,3] + 108.696;
   1:L PR[91] R[100]mm/sec CNT100;
   1:  PR[91,1] = PR[90,1] + 64.329;
   1:  PR[91,2] = PR[90,2] + -12.776;
   1:  PR[91,3] = PR[90,3] + 108.719;
   1:L PR[91] R[100]mm/sec CNT100;
   1:  PR[91,1] = PR[90,1] + 65.406;
   1:  PR[91,2] = PR[90,2] + -10.217;
   1:  PR[91,3] = PR[90,3] + 108.724;
   1:L PR[91] R[100]mm/sec CNT100;
   1:  PR[91,1] = PR[90,1] + 65.848;
   1:  PR[91,2] = PR[90,2] + -8.943;
   1:  PR[91,3] = PR[90,3] + 108.738;
   1:L PR[91] R[100]mm/sec CNT100;
   1:  PR[91,1] = PR[90,1] + 66.790;
   1:  PR[91,2] = PR[90,2] + -5.141;
   1:  PR[91,3] = PR[90,3] + 108.745;
   1:L PR[91] R[100]mm/sec CNT100;
   1:  PR[91,1] = PR[90,1] + 67.153;
   1:  PR[91,2] = PR[90,2] + -0.729;
   1:  PR[91,3] = PR[90,3] + 108.764;
   1:L PR[91] R[100]mm/sec CNT100;
   1:  PR[91,1] = PR[90,1] + 66.790;
   1:  PR[91,2] = PR[90,2] + 3.683;
   1:  PR[91,3] = PR[90,3] + 108.786;
   1:L PR[91] R[100]mm/sec CNT100;
   1:  PR[91,1] = PR[90,1] + 65.848;
   1:  PR[91,2] = PR[90,2] + 7.484;
   1:  PR[91,3] = PR[90,3] + 108.808;
   1:L PR[91] R[100]mm/sec CNT100;
   1:  PR[91,1] = PR[90,1] + 65.406;
   1:  PR[91,2] = PR[90,2] + 8.758;
   1:  PR[91,3] = PR[90,3] + 108.828;
   1:L PR[91] R[100]mm/sec CNT100;
   1:  PR[91,1] = PR[90,1] + 64.312;
   1:  PR[91,2] = PR[90,2] + 11.357;
   1:  PR[91,3] = PR[90,3] + 108.835;
   1:L PR[91] R[100]mm/sec CNT100;
   1:  PR[91,1] = PR[90,1] + 61.839;
   1:  PR[91,2] = PR[90,2] + 15.481;
   1:  PR[91,3] = PR[90,3] + 108.849;
   1:L PR[91] R[100]mm/sec CNT100;
   1:  PR[91,1] = PR[90,1] + 61.487;
   1:  PR[91,2] = PR[90,2] + 16.090;
   1:  PR[91,3] = PR[90,3] + 108.873;
   1:L PR[91] R[100]mm/sec CNT100;
   1:  PR[91,1] = PR[90,1] + 59.088;
   1:  PR[91,2] = PR[90,2] + 18.833;
   1:  PR[91,3] = PR[90,3] + 108.876;
   1:L PR[91] R[100]mm/sec CNT100;
   1:  PR[91,1] = PR[90,1] + 57.391;
   1:  PR[91,2] = PR[90,2] + 20.836;
   1:  PR[91,3] = PR[90,3] + 108.894;
   1:L PR[91] R[100]mm/sec CNT100;
   1:  PR[91,1] = PR[90,1] + 56.151;
   1:  PR[91,2] = PR[90,2] + 21.824;
   1:  PR[91,3] = PR[90,3] + 108.907;
   1:L PR[91] R[100]mm/sec CNT100;
   1:  PR[91,1] = PR[90,1] + 52.443;
   1:  PR[91,2] = PR[90,2] + 24.849;
   1:  PR[91,3] = PR[90,3] + 108.915;
   1:L PR[91] R[100]mm/sec CNT100;
   1:  PR[91,1] = PR[90,1] + 47.714;
   1:  PR[91,2] = PR[90,2] + 27.570;
   1:  PR[91,3] = PR[90,3] + 108.939;
   1:L PR[91] R[100]mm/sec CNT100;
   1:  PR[91,1] = PR[90,1] + 46.280;
   1:  PR[91,2] = PR[90,2] + 28.232;
   1:  PR[91,3] = PR[90,3] + 108.966;
   1:L PR[91] R[100]mm/sec CNT100;
   1:  PR[91,1] = PR[90,1] + 42.792;
   1:  PR[91,2] = PR[90,2] + 29.483;
   1:  PR[91,3] = PR[90,3] + 108.974;
   1:L PR[91] R[100]mm/sec CNT100;
   1:  PR[91,1] = PR[90,1] + 39.992;
   1:  PR[91,2] = PR[90,2] + 30.242;
   1:  PR[91,3] = PR[90,3] + 108.993;
   1:L PR[91] R[100]mm/sec CNT100;
   1:  PR[91,1] = PR[90,1] + 37.663;
   1:  PR[91,2] = PR[90,2] + 30.635;
   1:  PR[91,3] = PR[90,3] + 109.007;
   1:L PR[91] R[100]mm/sec CNT100;
   1:  PR[91,1] = PR[90,1] + 33.803;
   1:  PR[91,2] = PR[90,2] + 31.016;
   1:  PR[91,3] = PR[90,3] + 109.019;
   1:L PR[91] R[100]mm/sec CNT100;
   1:  PR[91,1] = PR[90,1] + 32.449;
   1:  PR[91,2] = PR[90,2] + 31.007;
   1:  PR[91,3] = PR[90,3] + 109.038;
   1:L PR[91] R[100]mm/sec CNT100;
   1:  PR[91,1] = PR[90,1] + 19.615;
   1:  PR[91,2] = PR[90,2] + 30.152;
   1:  PR[91,3] = PR[90,3] + 109.045;
   1:L PR[91] R[100]mm/sec CNT100;
   1:  PR[91,1] = PR[90,1] + 12.059;
   1:  PR[91,2] = PR[90,2] + 28.723;
   1:  PR[91,3] = PR[90,3] + 109.109;
   1:L PR[91] R[100]mm/sec CNT100;
   1:  PR[91,1] = PR[90,1] + 10.594;
   1:  PR[91,2] = PR[90,2] + 28.502;
   1:  PR[91,3] = PR[90,3] + 109.148;
   1:L PR[91] R[100]mm/sec CNT100;
   1:  PR[91,1] = PR[90,1] + 9.097;
   1:  PR[91,2] = PR[90,2] + 28.165;
   1:  PR[91,3] = PR[90,3] + 109.155;
   1:L PR[91] R[100]mm/sec CNT100;
   1:  PR[91,1] = PR[90,1] + 3.791;
   1:  PR[91,2] = PR[90,2] + 26.792;
   1:  PR[91,3] = PR[90,3] + 109.163;
   1:L PR[91] R[100]mm/sec CNT100;
   1:  PR[91,1] = PR[90,1] + 0.239;
   1:  PR[91,2] = PR[90,2] + 25.650;
   1:  PR[91,3] = PR[90,3] + 109.190;
   1:L PR[91] R[100]mm/sec CNT100;
   1:  PR[91,1] = PR[90,1] + -2.826;
   1:  PR[91,2] = PR[90,2] + 24.839;
   1:  PR[91,3] = PR[90,3] + 109.209;
   1:L PR[91] R[100]mm/sec CNT100;
   1:  PR[91,1] = PR[90,1] + -11.016;
   1:  PR[91,2] = PR[90,2] + 21.890;
   1:  PR[91,3] = PR[90,3] + 109.224;
   1:L PR[91] R[100]mm/sec CNT100;
   1:  PR[91,1] = PR[90,1] + -18.038;
   1:  PR[91,2] = PR[90,2] + 18.541;
   1:  PR[91,3] = PR[90,3] + 109.268;
   1:L PR[91] R[100]mm/sec CNT100;
   1:  PR[91,1] = PR[90,1] + -20.653;
   1:  PR[91,2] = PR[90,2] + 16.891;
   1:  PR[91,3] = PR[90,3] + 109.307;
   1:L PR[91] R[100]mm/sec CNT100;
   1:  PR[91,1] = PR[90,1] + -23.788;
   1:  PR[91,2] = PR[90,2] + 14.892;
   1:  PR[91,3] = PR[90,3] + 109.322;
   1:L PR[91] R[100]mm/sec CNT100;
   1:  PR[91,1] = PR[90,1] + -28.240;
   1:  PR[91,2] = PR[90,2] + 11.036;
   1:  PR[91,3] = PR[90,3] + 109.341;
   1:L PR[91] R[100]mm/sec CNT100;
   1:  PR[91,1] = PR[90,1] + -31.353;
   1:  PR[91,2] = PR[90,2] + 7.097;
   1:  PR[91,3] = PR[90,3] + 109.370;
   1:L PR[91] R[100]mm/sec CNT100;
   1:  PR[91] = PR[90];
   1:  PR[91,1] = PR[90,1] + -31.033;
   1:  PR[91,2] = PR[90,2] + 3.188;
   1:  PR[91,3] = PR[90,3] + 110.695;
   1:L PR[91] R[100]mm/sec CNT100;
   1:  PR[91,1] = PR[90,1] + -31.630;
   1:  PR[91,2] = PR[90,2] + -0.729;
   1:  PR[91,3] = PR[90,3] + 109.417;
   1:L PR[91] R[100]mm/sec CNT100;
   1:  PR[91,1] = PR[90,1] + -31.033;
   1:  PR[91,2] = PR[90,2] + -4.647;
   1:  PR[91,3] = PR[90,3] + 109.437;
   1:L PR[91] R[100]mm/sec CNT100;
   1:  PR[91,1] = PR[90,1] + -29.205;
   1:  PR[91,2] = PR[90,2] + -8.618;
   1:  PR[91,3] = PR[90,3] + 109.457;
   1:L PR[91] R[100]mm/sec CNT100;
   1:  PR[91,1] = PR[90,1] + -26.069;
   1:  PR[91,2] = PR[90,2] + -12.589;
   1:  PR[91,3] = PR[90,3] + 109.479;
   1:L PR[91] R[100]mm/sec CNT100;
   1:  PR[91,1] = PR[90,1] + -23.927;
   1:  PR[91,2] = PR[90,2] + -14.454;
   1:  PR[91,3] = PR[90,3] + 109.504;
   1:L PR[91] R[100]mm/sec CNT100;
   1:  PR[91,1] = PR[90,1] + -21.592;
   1:  PR[91,2] = PR[90,2] + -16.469;
   1:  PR[91,3] = PR[90,3] + 109.519;
   1:L PR[91] R[100]mm/sec CNT100;
   1:  PR[91,1] = PR[90,1] + -15.798;
   1:  PR[91,2] = PR[90,2] + -20.149;
   1:  PR[91,3] = PR[90,3] + 109.534;
   1:L PR[91] R[100]mm/sec CNT100;
   1:  PR[91,1] = PR[90,1] + -8.731;
   1:  PR[91,2] = PR[90,2] + -23.521;
   1:  PR[91,3] = PR[90,3] + 109.569;
   1:L PR[91] R[100]mm/sec CNT100;
   1:  PR[91,1] = PR[90,1] + -0.438;
   1:  PR[91,2] = PR[90,2] + -26.511;
   1:  PR[91,3] = PR[90,3] + 109.608;
   1:L PR[91] R[100]mm/sec CNT100;
   1:  PR[91,1] = PR[90,1] + 4.858;
   1:  PR[91,2] = PR[90,2] + -28.207;
   1:  PR[91,3] = PR[90,3] + 109.652;
   1:L PR[91] R[100]mm/sec CNT100;
   1:  PR[91,1] = PR[90,1] + 11.413;
   1:  PR[91,2] = PR[90,2] + -29.903;
   1:  PR[91,3] = PR[90,3] + 109.680;
   1:L PR[91] R[100]mm/sec CNT100;
   1:  PR[91,1] = PR[90,1] + 12.090;
   1:  PR[91,2] = PR[90,2] + -30.123;
   1:  PR[91,3] = PR[90,3] + 109.714;
   1:L PR[91] R[100]mm/sec CNT100;
   1:  PR[91,1] = PR[90,1] + 21.116;
   1:  PR[91,2] = PR[90,2] + -31.831;
   1:  PR[91,3] = PR[90,3] + 109.718;
   1:L PR[91] R[100]mm/sec CNT100;
   1:  PR[91,1] = PR[90,1] + 32.183;
   1:  PR[91,2] = PR[90,2] + -32.570;
   1:  PR[91,3] = PR[90,3] + 109.764;
   1:L PR[91] R[100]mm/sec CNT100;
   1:  PR[91,1] = PR[90,1] + 34.634;
   1:  PR[91,2] = PR[90,2] + -32.587;
   1:  PR[91,3] = PR[90,3] + 109.820;
   1:L PR[91] R[100]mm/sec CNT100;
   1:  PR[91,1] = PR[90,1] + 37.384;
   1:  PR[91,2] = PR[90,2] + -32.313;
   1:  PR[91,3] = PR[90,3] + 109.832;
   1:L PR[91] R[100]mm/sec CNT100;
   1:  PR[91,1] = PR[90,1] + 41.025;
   1:  PR[91,2] = PR[90,2] + -31.699;
   1:  PR[91,3] = PR[90,3] + 109.846;
   1:L PR[91] R[100]mm/sec CNT100;
   1:  PR[91,1] = PR[90,1] + 42.554;
   1:  PR[91,2] = PR[90,2] + -31.284;
   1:  PR[91,3] = PR[90,3] + 109.865;
   1:L PR[91] R[100]mm/sec CNT100;
   1:  PR[91,1] = PR[90,1] + 47.555;
   1:  PR[91,2] = PR[90,2] + -29.492;
   1:  PR[91,3] = PR[90,3] + 109.873;
   1:L PR[91] R[100]mm/sec CNT100;
   1:  PR[91,1] = PR[90,1] + 47.563;
   1:  PR[91,2] = PR[90,2] + -29.488;
   1:  PR[91,3] = PR[90,3] + 109.900;
   1:L PR[91] R[100]mm/sec CNT100;
   1:  PR[91,1] = PR[90,1] + 53.203;
   1:  PR[91,2] = PR[90,2] + -26.355;
   1:L PR[91] R[100]mm/sec CNT100;
   1:  PR[91,1] = PR[90,1] + 55.545;
   1:  PR[91,2] = PR[90,2] + -24.445;
   1:  PR[91,3] = PR[90,3] + 109.932;
   1:L PR[91] R[100]mm/sec CNT100;
   1:  PR[91,1] = PR[90,1] + 58.193;
   1:  PR[91,2] = PR[90,2] + -22.332;
   1:  PR[91,3] = PR[90,3] + 109.947;
   1:L PR[91] R[100]mm/sec CNT100;
   1:  PR[91,1] = PR[90,1] + 59.270;
   1:  PR[91,2] = PR[90,2] + -21.086;
   1:  PR[91,3] = PR[90,3] + 109.964;
   1:L PR[91] R[100]mm/sec CNT100;
   1:  PR[91,1] = PR[90,1] + 61.513;
   1:  PR[91,2] = PR[90,2] + -18.578;
   1:  PR[91,3] = PR[90,3] + 109.973;
   1:L PR[91] R[100]mm/sec CNT100;
   1:  PR[91,1] = PR[90,1] + 62.353;
   1:  PR[91,2] = PR[90,2] + -17.590;
   1:  PR[91,3] = PR[90,3] + 109.989;
   1:L PR[91] R[100]mm/sec CNT100;
   1:  PR[91,1] = PR[90,1] + 63.404;
   1:  PR[91,2] = PR[90,2] + -15.783;
   1:  PR[91,3] = PR[90,3] + 109.996;
   1:L PR[91] R[100]mm/sec CNT100;
   1:  PR[91,1] = PR[90,1] + 64.827;
   1:  PR[91,2] = PR[90,2] + -13.617;
   1:  PR[91,3] = PR[90,3] + 110.007;
   1:L PR[91] R[100]mm/sec CNT100;
   1:  PR[91,1] = PR[90,1] + 66.603;
   1:  PR[91,2] = PR[90,2] + -9.430;
   1:  PR[91,3] = PR[90,3] + 110.020;
   1:L PR[91] R[100]mm/sec CNT100;
   1:  PR[91,1] = PR[90,1] + 67.642;
   1:  PR[91,2] = PR[90,2] + -5.250;
   1:  PR[91,3] = PR[90,3] + 110.042;
   1:L PR[91] R[100]mm/sec CNT100;
   1:  PR[91,1] = PR[90,1] + 68.002;
   1:  PR[91,2] = PR[90,2] + -0.831;
   1:  PR[91,3] = PR[90,3] + 110.064;
   1:L PR[91] R[100]mm/sec CNT100;
   1:  PR[91,1] = PR[90,1] + 68.025;
   1:  PR[91,2] = PR[90,2] + -0.670;
   1:  PR[91,3] = PR[90,3] + 110.086;
   1:L PR[91] R[100]mm/sec CNT100;
   1:  PR[91,1] = PR[90,1] + 67.675;
   1:  PR[91,2] = PR[90,2] + 3.605;
   1:  PR[91,3] = PR[90,3] + 110.087;
   1:L PR[91] R[100]mm/sec CNT100;
   1:  PR[91,1] = PR[90,1] + 67.657;
   1:  PR[91,2] = PR[90,2] + 3.733;
   1:  PR[91,3] = PR[90,3] + 110.109;
   1:L PR[91] R[100]mm/sec CNT100;
   1:  PR[91,1] = PR[90,1] + 66.603;
   1:  PR[91,2] = PR[90,2] + 7.971;
   1:L PR[91] R[100]mm/sec CNT100;
   1:  PR[91,1] = PR[90,1] + 64.818;
   1:  PR[91,2] = PR[90,2] + 12.179;
   1:  PR[91,3] = PR[90,3] + 110.131;
   1:L PR[91] R[100]mm/sec CNT100;
   1:  PR[91,1] = PR[90,1] + 62.372;
   1:  PR[91,2] = PR[90,2] + 16.108;
   1:  PR[91,3] = PR[90,3] + 110.154;
   1:L PR[91] R[100]mm/sec CNT100;
   1:  PR[91,1] = PR[90,1] + 61.513;
   1:  PR[91,2] = PR[90,2] + 17.120;
   1:  PR[91,3] = PR[90,3] + 110.178;
   1:L PR[91] R[100]mm/sec CNT100;
   1:  PR[91,1] = PR[90,1] + 59.270;
   1:  PR[91,2] = PR[90,2] + 19.627;
   1:  PR[91,3] = PR[90,3] + 110.184;
   1:L PR[91] R[100]mm/sec CNT100;
   1:  PR[91,1] = PR[90,1] + 58.191;
   1:  PR[91,2] = PR[90,2] + 20.876;
   1:  PR[91,3] = PR[90,3] + 110.201;
   1:L PR[91] R[100]mm/sec CNT100;
   1:  PR[91,1] = PR[90,1] + 55.544;
   1:  PR[91,2] = PR[90,2] + 22.986;
   1:  PR[91,3] = PR[90,3] + 110.210;
   1:L PR[91] R[100]mm/sec CNT100;
   1:  PR[91,1] = PR[90,1] + 53.203;
   1:  PR[91,2] = PR[90,2] + 24.896;
   1:  PR[91,3] = PR[90,3] + 110.227;
   1:L PR[91] R[100]mm/sec CNT100;
   1:  PR[91,1] = PR[90,1] + 47.567;
   1:  PR[91,2] = PR[90,2] + 28.027;
   1:  PR[91,3] = PR[90,3] + 110.242;
   1:L PR[91] R[100]mm/sec CNT100;
   1:  PR[91,1] = PR[90,1] + 47.560;
   1:  PR[91,2] = PR[90,2] + 28.030;
   1:  PR[91,3] = PR[90,3] + 110.274;
   1:L PR[91] R[100]mm/sec CNT100;
   1:  PR[91,1] = PR[90,1] + 42.554;
   1:  PR[91,2] = PR[90,2] + 29.826;
   1:L PR[91] R[100]mm/sec CNT100;
   1:  PR[91,1] = PR[90,1] + 41.023;
   1:  PR[91,2] = PR[90,2] + 30.241;
   1:  PR[91,3] = PR[90,3] + 110.301;
   1:L PR[91] R[100]mm/sec CNT100;
   1:  PR[91,1] = PR[90,1] + 37.378;
   1:  PR[91,2] = PR[90,2] + 30.856;
   1:  PR[91,3] = PR[90,3] + 110.309;
   1:L PR[91] R[100]mm/sec CNT100;
   1:  PR[91,1] = PR[90,1] + 34.625;
   1:  PR[91,2] = PR[90,2] + 31.128;
   1:  PR[91,3] = PR[90,3] + 110.328;
   1:L PR[91] R[100]mm/sec CNT100;
   1:  PR[91,1] = PR[90,1] + 32.165;
   1:  PR[91,2] = PR[90,2] + 31.111;
   1:  PR[91,3] = PR[90,3] + 110.342;
   1:L PR[91] R[100]mm/sec CNT100;
   1:  PR[91,1] = PR[90,1] + 21.135;
   1:  PR[91,2] = PR[90,2] + 30.375;
   1:  PR[91,3] = PR[90,3] + 110.354;
   1:L PR[91] R[100]mm/sec CNT100;
   1:  PR[91,1] = PR[90,1] + 12.092;
   1:  PR[91,2] = PR[90,2] + 28.665;
   1:  PR[91,3] = PR[90,3] + 110.410;
   1:L PR[91] R[100]mm/sec CNT100;
   1:  PR[91,1] = PR[90,1] + 11.413;
   1:  PR[91,2] = PR[90,2] + 28.444;
   1:  PR[91,3] = PR[90,3] + 110.456;
   1:L PR[91] R[100]mm/sec CNT100;
   1:  PR[91,1] = PR[90,1] + 4.858;
   1:  PR[91,2] = PR[90,2] + 26.748;
   1:  PR[91,3] = PR[90,3] + 110.459;
   1:L PR[91] R[100]mm/sec CNT100;
   1:  PR[91,1] = PR[90,1] + -0.438;
   1:  PR[91,2] = PR[90,2] + 25.052;
   1:  PR[91,3] = PR[90,3] + 110.494;
   1:L PR[91] R[100]mm/sec CNT100;
   1:  PR[91,1] = PR[90,1] + -8.731;
   1:  PR[91,2] = PR[90,2] + 22.063;
   1:  PR[91,3] = PR[90,3] + 110.521;
   1:L PR[91] R[100]mm/sec CNT100;
   1:  PR[91,1] = PR[90,1] + -15.798;
